LIN {X 0,Y 122.403,Z 271.681,A -85,B 0,C 180,E1 -25569.931,E2 -25569.931} C_VEL
LIN {X 0,Y 122.203,Z 271.74,A -85,B 0,C 180,E1 -25573.312,E2 -25573.312} C_VEL
LIN {X 0,Y 122.006,Z 271.743,A -85,B 0,C 180,E1 -25580.233,E2 -25580.233} C_VEL
LIN {X 0,Y 121.968,Z 271.772,A -85,B 0,C 180,E1 -25583.801,E2 -25583.801} C_VEL
LIN {X 0,Y 121.949,Z 271.761,A -85,B 0,C 180,E1 -25590.17,E2 -25590.17} C_VEL
LIN {X 0,Y 121.983,Z 272.052,A -85,B 0,C 180,E1 -25592.462,E2 -25592.462} C_VEL
LIN {X 0,Y 122.24,Z 273.019,A -85,B 0,C 180,E1 -25593.12,E2 -25593.12} C_VEL
LIN {X 0,Y 123.846,Z 275.828,A -85,B 0,C 180,E1 -25594.219,E2 -25594.219} C_VEL
LIN {X 0,Y 125.183,Z 277.203,A -85,B 0,C 180,E1 -25594.99,E2 -25594.99} C_VEL
LIN {X 0,Y 127.179,Z 280.419,A -85,B 0,C 180,E1 -25596.188,E2 -25596.188} C_VEL
LIN {X 0,Y 128.715,Z 282.669,A -85,B 0,C 180,E1 -25597.05,E2 -25597.05} C_VEL
LIN {X 0,Y 133.456,Z 290.014,A -85,B 0,C 180,E1 -25599.546,E2 -25599.546} C_VEL
LIN {X 0,Y 138.65,Z 299.249,A -85,B 0,C 180,E1 -25602.083,E2 -25602.083} C_VEL
LIN {X 0,Y 142.571,Z 309.17,A -85,B 0,C 180,E1 -25604.02,E2 -25604.02} C_VEL
LIN {X 0,Y 147.025,Z 322.671,A -85,B 0,C 180,E1 -25606.191,E2 -25606.191} C_VEL
LIN {X 0,Y 147.183,Z 326.823,A -85,B 0,C 180,E1 -25606.489,E2 -25606.489} C_VEL
LIN {X 0,Y 144.077,Z 373.493,A -85,B 0,C 180,E1 -25608.588,E2 -25608.588} C_VEL
LIN {X 0,Y 142.334,Z 386.809,A -85,B 0,C 180,E1 -25609.647,E2 -25609.647} C_VEL
LIN {X 0,Y 140.104,Z 399.24,A -85,B 0,C 180,E1 -25611.163,E2 -25611.163} C_VEL
LIN {X 0,Y 137.46,Z 410.573,A -85,B 0,C 180,E1 -25613.071,E2 -25613.071} C_VEL
LIN {X 0,Y 134.929,Z 419.645,A -85,B 0,C 180,E1 -25615.038,E2 -25615.038} C_VEL
LIN {X 0,Y 131.957,Z 429.601,A -85,B 0,C 180,E1 -25617.813,E2 -25617.813} C_VEL
LIN {X 0,Y 128.677,Z 439.018,A -85,B 0,C 180,E1 -25621.144,E2 -25621.144} C_VEL
LIN {X 0,Y 126.257,Z 446.37,A -85,B 0,C 180,E1 -25624.438,E2 -25624.438} C_VEL
LIN {X 0,Y 123.386,Z 454.68,A -85,B 0,C 180,E1 -25629.14,E2 -25629.14} C_VEL
LIN {X 0,Y 121.564,Z 460.326,A -85,B 0,C 180,E1 -25633.193,E2 -25633.193} C_VEL
LIN {X 0,Y 120.15,Z 465.825,A -85,B 0,C 180,E1 -25638.181,E2 -25638.181} C_VEL
LIN {X 0,Y 119.423,Z 470.097,A -85,B 0,C 180,E1 -25643.235,E2 -25643.235} C_VEL
LIN {X 0,Y 119.243,Z 472.346,A -85,B 0,C 180,E1 -25646.616,E2 -25646.616} C_VEL
LIN {X 0,Y 119.301,Z 474.118,A -85,B 0,C 180,E1 -25649.995,E2 -25649.995} C_VEL
LIN {X 0,Y 119.243,Z 475.435,A -85,B 0,C 180,E1 -25653.374,E2 -25653.374} C_VEL
LIN {X 0,Y 119.973,Z 476.91,A -85,B 0,C 180,E1 -25660.116,E2 -25660.116} C_VEL
LIN {X 0,Y 120.788,Z 477.062,A -85,B 0,C 180,E1 -25663.453,E2 -25663.453} C_VEL
LIN {X 0,Y 123.519,Z 476.182,A -85,B 0,C 180,E1 -25669.956,E2 -25669.956} C_VEL
LIN {X 0,Y 127.871,Z 473.795,A -85,B 0,C 180,E1 -25676.079,E2 -25676.079} C_VEL
LIN {X 0,Y 132.095,Z 470.901,A -85,B 0,C 180,E1 -25680.355,E2 -25680.355} C_VEL
LIN {X 0,Y 137.033,Z 466.958,A -85,B 0,C 180,E1 -25684.4,E2 -25684.4} C_VEL
LIN {X 0,Y 142.426,Z 462.037,A -85,B 0,C 180,E1 -25688.078,E2 -25688.078} C_VEL
LIN {X 0,Y 148.475,Z 455.82,A -85,B 0,C 180,E1 -25691.499,E2 -25691.499} C_VEL
LIN {X 0,Y 152.037,Z 451.846,A -85,B 0,C 180,E1 -25693.187,E2 -25693.187} C_VEL
LIN {X 0,Y 153.514,Z 449.546,A -85,B 0,C 180,E1 -25694.277,E2 -25694.277} C_VEL
LIN {X 0,Y 155.933,Z 442.183,A -85,B 0,C 180,E1 -25698.383,E2 -25698.383} C_VEL
LIN {X 0,Y 157.534,Z 439.51,A -85,B 0,C 180,E1 -25699.288,E2 -25699.288} C_VEL
LIN {X 0,Y 163.973,Z 429.783,A -85,B 0,C 180,E1 -25701.456,E2 -25701.456} C_VEL
LIN {X 0,Y 170.017,Z 419.002,A -85,B 0,C 180,E1 -25703.21,E2 -25703.21} C_VEL
LIN {X 0,Y 175.47,Z 406.794,A -85,B 0,C 180,E1 -25704.686,E2 -25704.686} C_VEL
LIN {X 0,Y 179.465,Z 395.485,A -85,B 0,C 180,E1 -25705.679,E2 -25705.679} C_VEL
LIN {X 0,Y 182.83,Z 382.797,A -85,B 0,C 180,E1 -25706.459,E2 -25706.459} C_VEL
LIN {X 0,Y 185.096,Z 369.4,A -85,B 0,C 180,E1 -25706.986,E2 -25706.986} C_VEL
LIN {X 0,Y 186.027,Z 359.421,A -85,B 0,C 180,E1 -25707.359,E2 -25707.359} C_VEL
LIN {X 0,Y 183.427,Z 352.397,A -85,B 0,C 180,E1 -25710.038,E2 -25710.038} C_VEL
LIN {X 0,Y 180.664,Z 345.623,A -85,B 0,C 180,E1 -25713.403,E2 -25713.403} C_VEL
LIN {X 0,Y 178.531,Z 341.006,A -85,B 0,C 180,E1 -25716.548,E2 -25716.548} C_VEL
LIN {X 0,Y 177.003,Z 337.999,A -85,B 0,C 180,E1 -25719.316,E2 -25719.316} C_VEL
LIN {X 0,Y 175.209,Z 334.802,A -85,B 0,C 180,E1 -25724.285,E2 -25724.285} C_VEL
LIN {X 0,Y 174.993,Z 333.83,A -85,B 0,C 180,E1 -25725.558,E2 -25725.558} C_VEL
LIN {X 0,Y 174.576,Z 333.513,A -85,B 0,C 180,E1 -25730.725,E2 -25730.725} C_VEL
LIN {X 0,Y 175.407,Z 334.052,A -85,B 0,C 180,E1 -25735.276,E2 -25735.276} C_VEL
LIN {X 0,Y 176.87,Z 337.493,A -85,B 0,C 180,E1 -25739.595,E2 -25739.595} C_VEL
LIN {X 0,Y 177.65,Z 338.721,A -85,B 0,C 180,E1 -25741.069,E2 -25741.069} C_VEL
LIN {X 0,Y 179.573,Z 342.304,A -85,B 0,C 180,E1 -25744.164,E2 -25744.164} C_VEL
LIN {X 0,Y 182.057,Z 347.068,A -85,B 0,C 180,E1 -25747.381,E2 -25747.381} C_VEL
LIN {X 0,Y 184.322,Z 352.16,A -85,B 0,C 180,E1 -25749.883,E2 -25749.883} C_VEL
LIN {X 0,Y 186.256,Z 356.945,A -85,B 0,C 180,E1 -25751.795,E2 -25751.795} C_VEL
LIN {X 0,Y 184.328,Z 373.568,A -85,B 0,C 180,E1 -25752.362,E2 -25752.362} C_VEL
LIN {X 0,Y 181.73,Z 386.098,A -85,B 0,C 180,E1 -25752.999,E2 -25752.999} C_VEL
LIN {X 0,Y 177.786,Z 399.152,A -85,B 0,C 180,E1 -25753.996,E2 -25753.996} C_VEL
LIN {X 0,Y 173.022,Z 411.143,A -85,B 0,C 180,E1 -25755.284,E2 -25755.284} C_VEL
LIN {X 0,Y 167.29,Z 422.614,A -85,B 0,C 180,E1 -25756.966,E2 -25756.966} C_VEL
LIN {X 0,Y 160.799,Z 433.232,A -85,B 0,C 180,E1 -25759.076,E2 -25759.076} C_VEL
LIN {X 0,Y 154.773,Z 441.601,A -85,B 0,C 180,E1 -25761.289,E2 -25761.289} C_VEL
LIN {X 0,Y 148.126,Z 449.538,A -85,B 0,C 180,E1 -25764.041,E2 -25764.041} C_VEL
LIN {X 0,Y 140.778,Z 457.024,A -85,B 0,C 180,E1 -25767.62,E2 -25767.62} C_VEL
LIN {X 0,Y 134.12,Z 462.882,A -85,B 0,C 180,E1 -25771.587,E2 -25771.587} C_VEL
LIN {X 0,Y 127.366,Z 467.973,A -85,B 0,C 180,E1 -25776.642,E2 -25776.642} C_VEL
LIN {X 0,Y 122.243,Z 471.149,A -85,B 0,C 180,E1 -25781.643,E2 -25781.643} C_VEL
LIN {X 0,Y 119.474,Z 472.56,A -85,B 0,C 180,E1 -25785.106,E2 -25785.106} C_VEL
LIN {X 0,Y 117.087,Z 473.521,A -85,B 0,C 180,E1 -25788.688,E2 -25788.688} C_VEL
LIN {X 0,Y 115.063,Z 473.981,A -85,B 0,C 180,E1 -25792.539,E2 -25792.539} C_VEL
LIN {X 0,Y 113.602,Z 473.972,A -85,B 0,C 180,E1 -25796.173,E2 -25796.173} C_VEL
LIN {X 0,Y 112.308,Z 473.302,A -85,B 0,C 180,E1 -25801.141,E2 -25801.141} C_VEL
LIN {X 0,Y 111.542,Z 471.221,A -85,B 0,C 180,E1 -25807.794,E2 -25807.794} C_VEL
LIN {X 0,Y 111.803,Z 468.27,A -85,B 0,C 180,E1 -25813.574,E2 -25813.574} C_VEL
LIN {X 0,Y 112.709,Z 464.215,A -85,B 0,C 180,E1 -25819.224,E2 -25819.224} C_VEL
LIN {X 0,Y 114.241,Z 458.968,A -85,B 0,C 180,E1 -25824.711,E2 -25824.711} C_VEL
LIN {X 0,Y 116.441,Z 452.342,A -85,B 0,C 180,E1 -25830.005,E2 -25830.005} C_VEL
LIN {X 0,Y 119.479,Z 444.069,A -85,B 0,C 180,E1 -25835.045,E2 -25835.045} C_VEL
LIN {X 0,Y 122.529,Z 435.547,A -85,B 0,C 180,E1 -25839.081,E2 -25839.081} C_VEL
LIN {X 0,Y 125.838,Z 426.24,A -85,B 0,C 180,E1 -25842.504,E2 -25842.504} C_VEL
LIN {X 0,Y 129.091,Z 416.094,A -85,B 0,C 180,E1 -25845.396,E2 -25845.396} C_VEL
LIN {X 0,Y 132.092,Z 405.057,A -85,B 0,C 180,E1 -25847.819,E2 -25847.819} C_VEL
LIN {X 0,Y 134.949,Z 392.373,A -85,B 0,C 180,E1 -25849.878,E2 -25849.878} C_VEL
LIN {X 0,Y 137.118,Z 379.343,A -85,B 0,C 180,E1 -25851.348,E2 -25851.348} C_VEL
LIN {X 0,Y 138.593,Z 365.838,A -85,B 0,C 180,E1 -25852.288,E2 -25852.288} C_VEL
LIN {X 0,Y 141.572,Z 321.306,A -85,B 0,C 180,E1 -25854.321,E2 -25854.321} C_VEL
LIN {X 0,Y 138.053,Z 311.535,A -85,B 0,C 180,E1 -25856.101,E2 -25856.101} C_VEL
LIN {X 0,Y 133.083,Z 301.541,A -85,B 0,C 180,E1 -25858.579,E2 -25858.579} C_VEL
LIN {X 0,Y 126.471,Z 290.227,A -85,B 0,C 180,E1 -25862.157,E2 -25862.157} C_VEL
LIN {X 0,Y 120.762,Z 281.835,A -85,B 0,C 180,E1 -25865.641,E2 -25865.641} C_VEL
LIN {X 0,Y 118.642,Z 278.829,A -85,B 0,C 180,E1 -25867.062,E2 -25867.062} C_VEL
LIN {X 0,Y 117.859,Z 277.647,A -85,B 0,C 180,E1 -25867.618,E2 -25867.618} C_VEL
LIN {X 0,Y 115.795,Z 275.519,A -85,B 0,C 180,E1 -25869.05,E2 -25869.05} C_VEL
LIN {X 0,Y 114.906,Z 273.28,A -85,B 0,C 180,E1 -25870.113,E2 -25870.113} C_VEL
LIN {X 0,Y 114.82,Z 272.739,A -85,B 0,C 180,E1 -25871.018,E2 -25871.018} C_VEL
LIN {X 0,Y 114.755,Z 272.648,A -85,B 0,C 180,E1 -25877.669,E2 -25877.669} C_VEL
LIN {X 0,Y 114.771,Z 272.671,A -85,B 0,C 180,E1 -25882.763,E2 -25882.763} C_VEL
LIN {X 0,Y 114.83,Z 272.625,A -85,B 0,C 180,E1 -25888.975,E2 -25888.975} C_VEL
LIN {X 0,Y 114.896,Z 272.673,A -85,B 0,C 180,E1 -25896.58,E2 -25896.58} C_VEL
LIN {X 0,Y 114.965,Z 272.598,A -85,B 0,C 180,E1 -25902.217,E2 -25902.217} C_VEL
LIN {X 0,Y 115.31,Z 272.62,A -85,B 0,C 180,E1 -25909.479,E2 -25909.479} C_VEL
LIN {X 0,Y 115.487,Z 272.532,A -85,B 0,C 180,E1 -25916.525,E2 -25916.525} C_VEL
LIN {X 0,Y 115.956,Z 272.498,A -85,B 0,C 180,E1 -25920.013,E2 -25920.013} C_VEL
LIN {X 0,Y 115.356,Z 272.57,A -85,B 0,C 180,E1 -25927.012,E2 -25927.012} C_VEL
LIN {X 0,Y 115.219,Z 272.595,A -85,B 0,C 180,E1 -25932.568,E2 -25932.568} C_VEL
LIN {X 0,Y 114.983,Z 272.632,A -85,B 0,C 180,E1 -25937.808,E2 -25937.808} C_VEL
LIN {X 0,Y 114.931,Z 272.641,A -85,B 0,C 180,E1 -25943.461,E2 -25943.461} C_VEL
LIN {X 0,Y 114.904,Z 272.908,A -85,B 0,C 180,E1 -25948.372,E2 -25948.372} C_VEL
LIN {X 0,Y 115.209,Z 274.1,A -85,B 0,C 180,E1 -25949.225,E2 -25949.225} C_VEL
LIN {X 0,Y 116.985,Z 276.842,A -85,B 0,C 180,E1 -25950.626,E2 -25950.626} C_VEL
LIN {X 0,Y 118.483,Z 278.361,A -85,B 0,C 180,E1 -25951.635,E2 -25951.635} C_VEL
LIN {X 0,Y 120.642,Z 281.71,A -85,B 0,C 180,E1 -25953.117,E2 -25953.117} C_VEL
LIN {X 0,Y 121.817,Z 283.352,A -85,B 0,C 180,E1 -25953.869,E2 -25953.869} C_VEL
LIN {X 0,Y 126.872,Z 290.91,A -85,B 0,C 180,E1 -25956.905,E2 -25956.905} C_VEL
LIN {X 0,Y 133.463,Z 302.405,A -85,B 0,C 180,E1 -25960.457,E2 -25960.457} C_VEL
LIN {X 0,Y 137.115,Z 311.613,A -85,B 0,C 180,E1 -25962.416,E2 -25962.416} C_VEL
LIN {X 0,Y 141.44,Z 325.033,A -85,B 0,C 180,E1 -25964.709,E2 -25964.709} C_VEL
LIN {X 0,Y 138.165,Z 373.629,A -85,B 0,C 180,E1 -25966.999,E2 -25966.999} C_VEL
LIN {X 0,Y 136.379,Z 386.631,A -85,B 0,C 180,E1 -25968.057,E2 -25968.057} C_VEL
LIN {X 0,Y 134.123,Z 398.758,A -85,B 0,C 180,E1 -25969.57,E2 -25969.57} C_VEL
LIN {X 0,Y 131.352,Z 410.199,A -85,B 0,C 180,E1 -25971.532,E2 -25971.532} C_VEL
LIN {X 0,Y 128.697,Z 419.304,A -85,B 0,C 180,E1 -25973.562,E2 -25973.562} C_VEL
LIN {X 0,Y 125.567,Z 429.32,A -85,B 0,C 180,E1 -25976.442,E2 -25976.442} C_VEL
LIN {X 0,Y 122.067,Z 438.887,A -85,B 0,C 180,E1 -25979.962,E2 -25979.962} C_VEL
LIN {X 0,Y 119.873,Z 445.38,A -85,B 0,C 180,E1 -25982.97,E2 -25982.97} C_VEL
LIN {X 0,Y 116.755,Z 453.855,A -85,B 0,C 180,E1 -25987.895,E2 -25987.895} C_VEL
LIN {X 0,Y 114.441,Z 460.654,A -85,B 0,C 180,E1 -25993.034,E2 -25993.034} C_VEL
LIN {X 0,Y 112.818,Z 466.865,A -85,B 0,C 180,E1 -25999.223,E2 -25999.223} C_VEL
LIN {X 0,Y 112.212,Z 470.866,A -85,B 0,C 180,E1 -26004.604,E2 -26004.604} C_VEL
LIN {X 0,Y 112.22,Z 473.796,A -85,B 0,C 180,E1 -26009.994,E2 -26009.994} C_VEL
LIN {X 0,Y 112.154,Z 475.171,A -85,B 0,C 180,E1 -26013.587,E2 -26013.587} C_VEL
LIN {X 0,Y 112.972,Z 476.74,A -85,B 0,C 180,E1 -26020.75,E2 -26020.75} C_VEL
LIN {X 0,Y 115.178,Z 476.779,A -85,B 0,C 180,E1 -26027.758,E2 -26027.758} C_VEL
LIN {X 0,Y 118.965,Z 475.247,A -85,B 0,C 180,E1 -26034.421,E2 -26034.421} C_VEL
LIN {X 0,Y 124.442,Z 472.172,A -85,B 0,C 180,E1 -26040.543,E2 -26040.543} C_VEL
LIN {X 0,Y 129.381,Z 468.73,A -85,B 0,C 180,E1 -26044.769,E2 -26044.769} C_VEL
LIN {X 0,Y 134.895,Z 464.25,A -85,B 0,C 180,E1 -26048.69,E2 -26048.69} C_VEL
LIN {X 0,Y 142.17,Z 457.507,A -85,B 0,C 180,E1 -26052.815,E2 -26052.815} C_VEL
LIN {X 0,Y 149.058,Z 450.213,A -85,B 0,C 180,E1 -26055.968,E2 -26055.968} C_VEL
LIN {X 0,Y 156.292,Z 441.211,A -85,B 0,C 180,E1 -26058.862,E2 -26058.862} C_VEL
LIN {X 0,Y 157.534,Z 439.51,A -85,B 0,C 180,E1 -26059.288,E2 -26059.288} C_VEL
LIN {X 0,Y 160.137,Z 435.355,A -85,B 0,C 180,E1 -26060.469,E2 -26060.469} C_VEL
LIN {X 0,Y 163.166,Z 428.411,A -85,B 0,C 180,E1 -26062.738,E2 -26062.738} C_VEL
LIN {X 0,Y 165.973,Z 421.086,A -85,B 0,C 180,E1 -26064.83,E2 -26064.83} C_VEL
LIN {X 0,Y 168.136,Z 416.223,A -85,B 0,C 180,E1 -26065.725,E2 -26065.725} C_VEL
LIN {X 0,Y 172.963,Z 405.394,A -85,B 0,C 180,E1 -26066.928,E2 -26066.928} C_VEL
LIN {X 0,Y 177.071,Z 393.675,A -85,B 0,C 180,E1 -26067.893,E2 -26067.893} C_VEL
LIN {X 0,Y 180.496,Z 380.166,A -85,B 0,C 180,E1 -26068.636,E2 -26068.636} C_VEL
LIN {X 0,Y 182.557,Z 367.334,A -85,B 0,C 180,E1 -26069.081,E2 -26069.081} C_VEL
LIN {X 0,Y 182.952,Z 362.799,A -85,B 0,C 180,E1 -26069.275,E2 -26069.275} C_VEL
LIN {X 0,Y 180.739,Z 356.713,A -85,B 0,C 180,E1 -26071.861,E2 -26071.861} C_VEL
LIN {X 0,Y 178.612,Z 351.184,A -85,B 0,C 180,E1 -26074.814,E2 -26074.814} C_VEL
LIN {X 0,Y 176.995,Z 347.376,A -85,B 0,C 180,E1 -26077.474,E2 -26077.474} C_VEL
LIN {X 0,Y 175.737,Z 344.777,A -85,B 0,C 180,E1 -26079.952,E2 -26079.952} C_VEL
LIN {X 0,Y 174.126,Z 341.381,A -85,B 0,C 180,E1 -26085.119,E2 -26085.119} C_VEL
LIN {X 0,Y 174.003,Z 340.799,A -85,B 0,C 180,E1 -26085.967,E2 -26085.967} C_VEL
LIN {X 0,Y 173.971,Z 340.663,A -85,B 0,C 180,E1 -26093.03,E2 -26093.03} C_VEL
LIN {X 0,Y 174.388,Z 341.072,A -85,B 0,C 180,E1 -26094.918,E2 -26094.918} C_VEL
LIN {X 0,Y 175.915,Z 344.609,A -85,B 0,C 180,E1 -26099.558,E2 -26099.558} C_VEL
LIN {X 0,Y 177.962,Z 348.626,A -85,B 0,C 180,E1 -26103.247,E2 -26103.247} C_VEL
LIN {X 0,Y 180.32,Z 353.423,A -85,B 0,C 180,E1 -26106.543,E2 -26106.543} C_VEL
LIN {X 0,Y 182.873,Z 359.659,A -85,B 0,C 180,E1 -26109.56,E2 -26109.56} C_VEL
LIN {X 0,Y 183.179,Z 360.526,A -85,B 0,C 180,E1 -26109.895,E2 -26109.895} C_VEL
LIN {X 0,Y 181.29,Z 375.016,A -85,B 0,C 180,E1 -26110.377,E2 -26110.377} C_VEL
LIN {X 0,Y 178.531,Z 387.326,A -85,B 0,C 180,E1 -26111.007,E2 -26111.007} C_VEL
LIN {X 0,Y 174.297,Z 400.567,A -85,B 0,C 180,E1 -26112.018,E2 -26112.018} C_VEL
LIN {X 0,Y 169.637,Z 411.763,A -85,B 0,C 180,E1 -26113.214,E2 -26113.214} C_VEL
LIN {X 0,Y 163.996,Z 422.64,A -85,B 0,C 180,E1 -26114.776,E2 -26114.776} C_VEL
LIN {X 0,Y 157.001,Z 433.645,A -85,B 0,C 180,E1 -26116.912,E2 -26116.912} C_VEL
LIN {X 0,Y 150.367,Z 442.437,A -85,B 0,C 180,E1 -26119.231,E2 -26119.231} C_VEL
LIN {X 0,Y 143.809,Z 449.846,A -85,B 0,C 180,E1 -26121.806,E2 -26121.806} C_VEL
LIN {X 0,Y 136.11,Z 457.281,A -85,B 0,C 180,E1 -26125.375,E2 -26125.375} C_VEL
LIN {X 0,Y 129.035,Z 463.133,A -85,B 0,C 180,E1 -26129.383,E2 -26129.383} C_VEL
LIN {X 0,Y 122.695,Z 467.622,A -85,B 0,C 180,E1 -26133.853,E2 -26133.853} C_VEL
LIN {X 0,Y 117.172,Z 470.875,A -85,B 0,C 180,E1 -26138.772,E2 -26138.772} C_VEL
LIN {X 0,Y 113.581,Z 472.578,A -85,B 0,C 180,E1 -26142.873,E2 -26142.873} C_VEL
LIN {X 0,Y 109.052,Z 474.029,A -85,B 0,C 180,E1 -26149.883,E2 -26149.883} C_VEL
LIN {X 0,Y 107.247,Z 474.118,A -85,B 0,C 180,E1 -26153.866,E2 -26153.866} C_VEL
LIN {X 0,Y 105.372,Z 473.395,A -85,B 0,C 180,E1 -26160.086,E2 -26160.086} C_VEL
LIN {X 0,Y 104.506,Z 471.675,A -85,B 0,C 180,E1 -26166.21,E2 -26166.21} C_VEL
LIN {X 0,Y 104.569,Z 468.88,A -85,B 0,C 180,E1 -26172.402,E2 -26172.402} C_VEL
LIN {X 0,Y 105.427,Z 464.981,A -85,B 0,C 180,E1 -26178.47,E2 -26178.47} C_VEL
LIN {X 0,Y 106.943,Z 459.901,A -85,B 0,C 180,E1 -26184.349,E2 -26184.349} C_VEL
LIN {X 0,Y 109.072,Z 453.516,A -85,B 0,C 180,E1 -26190.006,E2 -26190.006} C_VEL
LIN {X 0,Y 112.176,Z 445.493,A -85,B 0,C 180,E1 -26195.4,E2 -26195.4} C_VEL
LIN {X 0,Y 115.39,Z 437.259,A -85,B 0,C 180,E1 -26199.647,E2 -26199.647} C_VEL
LIN {X 0,Y 119.136,Z 427.186,A -85,B 0,C 180,E1 -26203.654,E2 -26203.654} C_VEL
LIN {X 0,Y 122.515,Z 417.27,A -85,B 0,C 180,E1 -26206.673,E2 -26206.673} C_VEL
LIN {X 0,Y 125.684,Z 406.532,A -85,B 0,C 180,E1 -26209.184,E2 -26209.184} C_VEL
LIN {X 0,Y 128.518,Z 394.802,A -85,B 0,C 180,E1 -26211.235,E2 -26211.235} C_VEL
LIN {X 0,Y 131.06,Z 381.118,A -85,B 0,C 180,E1 -26212.921,E2 -26212.921} C_VEL
LIN {X 0,Y 132.678,Z 367.926,A -85,B 0,C 180,E1 -26213.93,E2 -26213.93} C_VEL
LIN {X 0,Y 135.961,Z 323.313,A -85,B 0,C 180,E1 -26215.99,E2 -26215.99} C_VEL
LIN {X 0,Y 132.938,Z 314.805,A -85,B 0,C 180,E1 -26217.661,E2 -26217.661} C_VEL
LIN {X 0,Y 128.25,Z 305.355,A -85,B 0,C 180,E1 -26220.189,E2 -26220.189} C_VEL
LIN {X 0,Y 122.378,Z 295.105,A -85,B 0,C 180,E1 -26223.653,E2 -26223.653} C_VEL
LIN {X 0,Y 117.429,Z 287.522,A -85,B 0,C 180,E1 -26226.913,E2 -26226.913} C_VEL
LIN {X 0,Y 114.355,Z 283.287,A -85,B 0,C 180,E1 -26229.148,E2 -26229.148} C_VEL
LIN {X 0,Y 112.028,Z 280.176,A -85,B 0,C 180,E1 -26230.99,E2 -26230.99} C_VEL
LIN {X 0,Y 111.299,Z 278.889,A -85,B 0,C 180,E1 -26231.635,E2 -26231.635} C_VEL
LIN {X 0,Y 108.763,Z 276.543,A -85,B 0,C 180,E1 -26233.771,E2 -26233.771} C_VEL
LIN {X 0,Y 107.719,Z 274.073,A -85,B 0,C 180,E1 -26235.222,E2 -26235.222} C_VEL
LIN {X 0,Y 107.688,Z 273.578,A -85,B 0,C 180,E1 -26236.77,E2 -26236.77} C_VEL
LIN {X 0,Y 107.699,Z 273.569,A -85,B 0,C 180,E1 -26244.053,E2 -26244.053} C_VEL
LIN {X 0,Y 107.768,Z 273.505,A -85,B 0,C 180,E1 -26248.571,E2 -26248.571} C_VEL
LIN {X 0,Y 107.863,Z 273.548,A -85,B 0,C 180,E1 -26257.004,E2 -26257.004} C_VEL
LIN {X 0,Y 107.86,Z 273.489,A -85,B 0,C 180,E1 -26261.003,E2 -26261.003} C_VEL
LIN {X 0,Y 108.228,Z 273.495,A -85,B 0,C 180,E1 -26268.781,E2 -26268.781} C_VEL
LIN {X 0,Y 108.291,Z 273.46,A -85,B 0,C 180,E1 -26272.557,E2 -26272.557} C_VEL
LIN {X 0,Y 108.886,Z 273.375,A -85,B 0,C 180,E1 -26280.014,E2 -26280.014} C_VEL
LIN {X 0,Y 108.297,Z 273.443,A -85,B 0,C 180,E1 -26287.472,E2 -26287.472} C_VEL
LIN {X 0,Y 108.153,Z 273.477,A -85,B 0,C 180,E1 -26292.884,E2 -26292.884} C_VEL
LIN {X 0,Y 107.897,Z 273.498,A -85,B 0,C 180,E1 -26301.007,E2 -26301.007} C_VEL
LIN {X 0,Y 107.937,Z 273.848,A -85,B 0,C 180,E1 -26303.567,E2 -26303.567} C_VEL
LIN {X 0,Y 108.215,Z 275.116,A -85,B 0,C 180,E1 -26304.432,E2 -26304.432} C_VEL
LIN {X 0,Y 109.831,Z 277.695,A -85,B 0,C 180,E1 -26305.995,E2 -26305.995} C_VEL
LIN {X 0,Y 111.72,Z 279.308,A -85,B 0,C 180,E1 -26307.529,E2 -26307.529} C_VEL
LIN {X 0,Y 113.783,Z 282.572,A -85,B 0,C 180,E1 -26309.246,E2 -26309.246} C_VEL
LIN {X 0,Y 115.207,Z 284.265,A -85,B 0,C 180,E1 -26310.304,E2 -26310.304} C_VEL
LIN {X 0,Y 120.719,Z 292.539,A -85,B 0,C 180,E1 -26314.133,E2 -26314.133} C_VEL
LIN {X 0,Y 125.969,Z 301.247,A -85,B 0,C 180,E1 -26317.345,E2 -26317.345} C_VEL
LIN {X 0,Y 129.654,Z 308.507,A -85,B 0,C 180,E1 -26319.45,E2 -26319.45} C_VEL
LIN {X 0,Y 133.071,Z 318.038,A -85,B 0,C 180,E1 -26321.451,E2 -26321.451} C_VEL
LIN {X 0,Y 135.778,Z 326.645,A -85,B 0,C 180,E1 -26323.008,E2 -26323.008} C_VEL
LIN {X 0,Y 132.451,Z 373.031,A -85,B 0,C 180,E1 -26325.218,E2 -26325.218} C_VEL
LIN {X 0,Y 130.604,Z 386.006,A -85,B 0,C 180,E1 -26326.273,E2 -26326.273} C_VEL
LIN {X 0,Y 128.036,Z 399.42,A -85,B 0,C 180,E1 -26328.005,E2 -26328.005} C_VEL
LIN {X 0,Y 124.845,Z 411.421,A -85,B 0,C 180,E1 -26330.177,E2 -26330.177} C_VEL
LIN {X 0,Y 122.153,Z 420.348,A -85,B 0,C 180,E1 -26332.31,E2 -26332.31} C_VEL
LIN {X 0,Y 118.889,Z 430.129,A -85,B 0,C 180,E1 -26335.315,E2 -26335.315} C_VEL
LIN {X 0,Y 115.016,Z 440.25,A -85,B 0,C 180,E1 -26339.33,E2 -26339.33} C_VEL
LIN {X 0,Y 112.267,Z 447.423,A -85,B 0,C 180,E1 -26343.003,E2 -26343.003} C_VEL
LIN {X 0,Y 109.178,Z 455.518,A -85,B 0,C 180,E1 -26348.27,E2 -26348.27} C_VEL
LIN {X 0,Y 107.303,Z 460.981,A -85,B 0,C 180,E1 -26352.852,E2 -26352.852} C_VEL
LIN {X 0,Y 105.838,Z 466.306,A -85,B 0,C 180,E1 -26358.503,E2 -26358.503} C_VEL
LIN {X 0,Y 105.134,Z 470.415,A -85,B 0,C 180,E1 -26364.239,E2 -26364.239} C_VEL
LIN {X 0,Y 105.128,Z 473.439,A -85,B 0,C 180,E1 -26369.994,E2 -26369.994} C_VEL
LIN {X 0,Y 105.089,Z 474.905,A -85,B 0,C 180,E1 -26373.829,E2 -26373.829} C_VEL
LIN {X 0,Y 105.998,Z 476.57,A -85,B 0,C 180,E1 -26381.467,E2 -26381.467} C_VEL
LIN {X 0,Y 108.428,Z 476.73,A -85,B 0,C 180,E1 -26388.904,E2 -26388.904} C_VEL
LIN {X 0,Y 110.223,Z 476.219,A -85,B 0,C 180,E1 -26392.487,E2 -26392.487} C_VEL
LIN {X 0,Y 115.286,Z 474.03,A -85,B 0,C 180,E1 -26399.183,E2 -26399.183} C_VEL
LIN {X 0,Y 120.028,Z 471.342,A -85,B 0,C 180,E1 -26403.79,E2 -26403.79} C_VEL
LIN {X 0,Y 126.973,Z 466.639,A -85,B 0,C 180,E1 -26408.983,E2 -26408.983} C_VEL
LIN {X 0,Y 133.696,Z 461.136,A -85,B 0,C 180,E1 -26413.101,E2 -26413.101} C_VEL
LIN {X 0,Y 140.591,Z 454.726,A -85,B 0,C 180,E1 -26416.449,E2 -26416.449} C_VEL
LIN {X 0,Y 147.978,Z 446.776,A -85,B 0,C 180,E1 -26419.448,E2 -26419.448} C_VEL
LIN {X 0,Y 154.41,Z 438.703,A -85,B 0,C 180,E1 -26421.726,E2 -26421.726} C_VEL
LIN {X 0,Y 160.385,Z 429.953,A -85,B 0,C 180,E1 -26423.621,E2 -26423.621} C_VEL
LIN {X 0,Y 166.618,Z 419.248,A -85,B 0,C 180,E1 -26425.33,E2 -26425.33} C_VEL
LIN {X 0,Y 168.136,Z 416.223,A -85,B 0,C 180,E1 -26425.725,E2 -26425.725} C_VEL
LIN {X 0,Y 170.201,Z 411.242,A -85,B 0,C 180,E1 -26426.557,E2 -26426.557} C_VEL
LIN {X 0,Y 172.468,Z 403.032,A -85,B 0,C 180,E1 -26428.27,E2 -26428.27} C_VEL
LIN {X 0,Y 174.356,Z 394.49,A -85,B 0,C 180,E1 -26429.785,E2 -26429.785} C_VEL
LIN {X 0,Y 175.74,Z 389.002,A -85,B 0,C 180,E1 -26430.31,E2 -26430.31} C_VEL
LIN {X 0,Y 178.689,Z 376.276,A -85,B 0,C 180,E1 -26430.885,E2 -26430.885} C_VEL
LIN {X 0,Y 180.094,Z 366.402,A -85,B 0,C 180,E1 -26431.24,E2 -26431.24} C_VEL
LIN {X 0,Y 177.797,Z 359.666,A -85,B 0,C 180,E1 -26434.454,E2 -26434.454} C_VEL
LIN {X 0,Y 175.986,Z 354.801,A -85,B 0,C 180,E1 -26437.514,E2 -26437.514} C_VEL
LIN {X 0,Y 174.551,Z 351.613,A -85,B 0,C 180,E1 -26440.507,E2 -26440.507} C_VEL
LIN {X 0,Y 173.085,Z 348.039,A -85,B 0,C 180,E1 -26445.891,E2 -26445.891} C_VEL
LIN {X 0,Y 172.783,Z 347.621,A -85,B 0,C 180,E1 -26448.257,E2 -26448.257} C_VEL
LIN {X 0,Y 173.294,Z 347.843,A -85,B 0,C 180,E1 -26454.131,E2 -26454.131} C_VEL
LIN {X 0,Y 175.111,Z 352.223,A -85,B 0,C 180,E1 -26459.882,E2 -26459.882} C_VEL
LIN {X 0,Y 176.701,Z 355.665,A -85,B 0,C 180,E1 -26462.837,E2 -26462.837} C_VEL
LIN {X 0,Y 178.814,Z 360.162,A -85,B 0,C 180,E1 -26465.943,E2 -26465.943} C_VEL
LIN {X 0,Y 180.259,Z 364.22,A -85,B 0,C 180,E1 -26467.874,E2 -26467.874} C_VEL
LIN {X 0,Y 178.452,Z 376.563,A -85,B 0,C 180,E1 -26468.337,E2 -26468.337} C_VEL
LIN {X 0,Y 175.037,Z 390.351,A -85,B 0,C 180,E1 -26469.069,E2 -26469.069} C_VEL
LIN {X 0,Y 170.819,Z 402.508,A -85,B 0,C 180,E1 -26470.008,E2 -26470.008} C_VEL
LIN {X 0,Y 165.691,Z 413.914,A -85,B 0,C 180,E1 -26471.245,E2 -26471.245} C_VEL
LIN {X 0,Y 159.642,Z 424.797,A -85,B 0,C 180,E1 -26472.847,E2 -26472.847} C_VEL
LIN {X 0,Y 152.692,Z 435.097,A -85,B 0,C 180,E1 -26474.875,E2 -26474.875} C_VEL
LIN {X 0,Y 145.379,Z 444.109,A -85,B 0,C 180,E1 -26477.315,E2 -26477.315} C_VEL
LIN {X 0,Y 136.98,Z 452.806,A -85,B 0,C 180,E1 -26480.568,E2 -26480.568} C_VEL
LIN {X 0,Y 129.089,Z 459.65,A -85,B 0,C 180,E1 -26484.241,E2 -26484.241} C_VEL
LIN {X 0,Y 122.56,Z 464.524,A -85,B 0,C 180,E1 -26488,E2 -26488} C_VEL
LIN {X 0,Y 115.143,Z 469.132,A -85,B 0,C 180,E1 -26493.304,E2 -26493.304} C_VEL
LIN {X 0,Y 108.912,Z 472.224,A -85,B 0,C 180,E1 -26499.264,E2 -26499.264} C_VEL
LIN {X 0,Y 105.811,Z 473.351,A -85,B 0,C 180,E1 -26503.07,E2 -26503.07} C_VEL
LIN {X 0,Y 102.012,Z 474.191,A -85,B 0,C 180,E1 -26509.247,E2 -26509.247} C_VEL
LIN {X 0,Y 99.389,Z 473.983,A -85,B 0,C 180,E1 -26515.557,E2 -26515.557} C_VEL
LIN {X 0,Y 98.265,Z 473.27,A -85,B 0,C 180,E1 -26519.965,E2 -26519.965} C_VEL
LIN {X 0,Y 97.543,Z 472.124,A -85,B 0,C 180,E1 -26524.394,E2 -26524.394} C_VEL
LIN {X 0,Y 97.364,Z 470.078,A -85,B 0,C 180,E1 -26529.728,E2 -26529.728} C_VEL
LIN {X 0,Y 97.812,Z 467.098,A -85,B 0,C 180,E1 -26535.442,E2 -26535.442} C_VEL
LIN {X 0,Y 99.224,Z 462.119,A -85,B 0,C 180,E1 -26542.437,E2 -26542.437} C_VEL
LIN {X 0,Y 101.343,Z 455.796,A -85,B 0,C 180,E1 -26549.013,E2 -26549.013} C_VEL
LIN {X 0,Y 104.289,Z 448.301,A -85,B 0,C 180,E1 -26554.838,E2 -26554.838} C_VEL
LIN {X 0,Y 107.623,Z 440.471,A -85,B 0,C 180,E1 -26559.491,E2 -26559.491} C_VEL
LIN {X 0,Y 111.267,Z 431.346,A -85,B 0,C 180,E1 -26563.707,E2 -26563.707} C_VEL
LIN {X 0,Y 115.153,Z 421.026,A -85,B 0,C 180,E1 -26567.315,E2 -26567.315} C_VEL
LIN {X 0,Y 118.842,Z 409.54,A -85,B 0,C 180,E1 -26570.336,E2 -26570.336} C_VEL
LIN {X 0,Y 122.083,Z 397.55,A -85,B 0,C 180,E1 -26572.667,E2 -26572.667} C_VEL
LIN {X 0,Y 124.801,Z 384.618,A -85,B 0,C 180,E1 -26574.431,E2 -26574.431} C_VEL
LIN {X 0,Y 126.784,Z 370.797,A -85,B 0,C 180,E1 -26575.662,E2 -26575.662} C_VEL
LIN {X 0,Y 130.338,Z 324.861,A -85,B 0,C 180,E1 -26577.888,E2 -26577.888} C_VEL
LIN {X 0,Y 127.752,Z 317.8,A -85,B 0,C 180,E1 -26579.426,E2 -26579.426} C_VEL
LIN {X 0,Y 122.98,Z 308.092,A -85,B 0,C 180,E1 -26582.262,E2 -26582.262} C_VEL
LIN {X 0,Y 118.236,Z 299.765,A -85,B 0,C 180,E1 -26585.324,E2 -26585.324} C_VEL
LIN {X 0,Y 113.614,Z 292.543,A -85,B 0,C 180,E1 -26588.658,E2 -26588.658} C_VEL
LIN {X 0,Y 110.804,Z 288.558,A -85,B 0,C 180,E1 -26590.905,E2 -26590.905} C_VEL
LIN {X 0,Y 108.167,Z 284.768,A -85,B 0,C 180,E1 -26593.246,E2 -26593.246} C_VEL
LIN {X 0,Y 105.657,Z 281.989,A -85,B 0,C 180,E1 -26595.585,E2 -26595.585} C_VEL
LIN {X 0,Y 104.713,Z 280.046,A -85,B 0,C 180,E1 -26596.654,E2 -26596.654} C_VEL
LIN {X 0,Y 101.89,Z 277.693,A -85,B 0,C 180,E1 -26599.675,E2 -26599.675} C_VEL
LIN {X 0,Y 100.731,Z 275.009,A -85,B 0,C 180,E1 -26601.763,E2 -26601.763} C_VEL
LIN {X 0,Y 100.653,Z 274.475,A -85,B 0,C 180,E1 -26603.615,E2 -26603.615} C_VEL
LIN {X 0,Y 100.672,Z 274.403,A -85,B 0,C 180,E1 -26606.912,E2 -26606.912} C_VEL
LIN {X 0,Y 100.721,Z 274.422,A -85,B 0,C 180,E1 -26615.268,E2 -26615.268} C_VEL
LIN {X 0,Y 100.774,Z 274.384,A -85,B 0,C 180,E1 -26619.609,E2 -26619.609} C_VEL
LIN {X 0,Y 101.127,Z 274.36,A -85,B 0,C 180,E1 -26627.982,E2 -26627.982} C_VEL
LIN {X 0,Y 101.228,Z 274.344,A -85,B 0,C 180,E1 -26632.034,E2 -26632.034} C_VEL
LIN {X 0,Y 101.817,Z 274.252,A -85,B 0,C 180,E1 -26640.015,E2 -26640.015} C_VEL
LIN {X 0,Y 101.232,Z 274.317,A -85,B 0,C 180,E1 -26647.997,E2 -26647.997} C_VEL
LIN {X 0,Y 101.024,Z 274.382,A -85,B 0,C 180,E1 -26654.19,E2 -26654.19} C_VEL
LIN {X 0,Y 100.916,Z 274.723,A -85,B 0,C 180,E1 -26656.971,E2 -26656.971} C_VEL
LIN {X 0,Y 101.205,Z 275.903,A -85,B 0,C 180,E1 -26658.094,E2 -26658.094} C_VEL
LIN {X 0,Y 102.866,Z 278.531,A -85,B 0,C 180,E1 -26660.251,E2 -26660.251} C_VEL
LIN {X 0,Y 104.953,Z 280.162,A -85,B 0,C 180,E1 -26662.402,E2 -26662.402} C_VEL
LIN {X 0,Y 106.713,Z 283.28,A -85,B 0,C 180,E1 -26664.277,E2 -26664.277} C_VEL
LIN {X 0,Y 108.88,Z 285.571,A -85,B 0,C 180,E1 -26666.21,E2 -26666.21} C_VEL
LIN {X 0,Y 112.39,Z 290.724,A -85,B 0,C 180,E1 -26669.211,E2 -26669.211} C_VEL
LIN {X 0,Y 116.926,Z 297.608,A -85,B 0,C 180,E1 -26672.598,E2 -26672.598} C_VEL
LIN {X 0,Y 122.07,Z 306.53,A -85,B 0,C 180,E1 -26676.013,E2 -26676.013} C_VEL
LIN {X 0,Y 125.122,Z 312.759,A -85,B 0,C 180,E1 -26677.907,E2 -26677.907} C_VEL
LIN {X 0,Y 128.173,Z 321.75,A -85,B 0,C 180,E1 -26679.875,E2 -26679.875} C_VEL
LIN {X 0,Y 130.173,Z 328.184,A -85,B 0,C 180,E1 -26681.128,E2 -26681.128} C_VEL
LIN {X 0,Y 126.756,Z 373.362,A -85,B 0,C 180,E1 -26683.341,E2 -26683.341} C_VEL
LIN {X 0,Y 124.734,Z 386.929,A -85,B 0,C 180,E1 -26684.505,E2 -26684.505} C_VEL
LIN {X 0,Y 122.285,Z 398.942,A -85,B 0,C 180,E1 -26686.105,E2 -26686.105} C_VEL
LIN {X 0,Y 118.943,Z 411.054,A -85,B 0,C 180,E1 -26688.332,E2 -26688.332} C_VEL
LIN {X 0,Y 116.101,Z 420.028,A -85,B 0,C 180,E1 -26690.529,E2 -26690.529} C_VEL
LIN {X 0,Y 112.65,Z 429.848,A -85,B 0,C 180,E1 -26693.646,E2 -26693.646} C_VEL
LIN {X 0,Y 108.507,Z 440.121,A -85,B 0,C 180,E1 -26697.892,E2 -26697.892} C_VEL
LIN {X 0,Y 105.956,Z 446.446,A -85,B 0,C 180,E1 -26701.25,E2 -26701.25} C_VEL
LIN {X 0,Y 102.595,Z 454.694,A -85,B 0,C 180,E1 -26706.797,E2 -26706.797} C_VEL
LIN {X 0,Y 100.5,Z 460.286,A -85,B 0,C 180,E1 -26711.652,E2 -26711.652} C_VEL
LIN {X 0,Y 98.887,Z 465.733,A -85,B 0,C 180,E1 -26717.683,E2 -26717.683} C_VEL
LIN {X 0,Y 98.078,Z 469.952,A -85,B 0,C 180,E1 -26723.823,E2 -26723.823} C_VEL
LIN {X 0,Y 98.028,Z 473.078,A -85,B 0,C 180,E1 -26729.994,E2 -26729.994} C_VEL
LIN {X 0,Y 98.015,Z 474.606,A -85,B 0,C 180,E1 -26734.105,E2 -26734.105} C_VEL
LIN {X 0,Y 98.297,Z 475.712,A -85,B 0,C 180,E1 -26738.215,E2 -26738.215} C_VEL
LIN {X 0,Y 100.138,Z 476.713,A -85,B 0,C 180,E1 -26746.297,E2 -26746.297} C_VEL
LIN {X 0,Y 103.675,Z 476.228,A -85,B 0,C 180,E1 -26753.993,E2 -26753.993} C_VEL
LIN {X 0,Y 109.145,Z 474.16,A -85,B 0,C 180,E1 -26760.999,E2 -26760.999} C_VEL
LIN {X 0,Y 116.058,Z 470.519,A -85,B 0,C 180,E1 -26767.262,E2 -26767.262} C_VEL
LIN {X 0,Y 122.454,Z 466.334,A -85,B 0,C 180,E1 -26771.729,E2 -26771.729} C_VEL
LIN {X 0,Y 128.627,Z 461.629,A -85,B 0,C 180,E1 -26775.252,E2 -26775.252} C_VEL
LIN {X 0,Y 135.828,Z 455.387,A -85,B 0,C 180,E1 -26778.605,E2 -26778.605} C_VEL
LIN {X 0,Y 143.508,Z 447.602,A -85,B 0,C 180,E1 -26781.58,E2 -26781.58} C_VEL
LIN {X 0,Y 150.15,Z 439.714,A -85,B 0,C 180,E1 -26783.836,E2 -26783.836} C_VEL
LIN {X 0,Y 156.318,Z 431.182,A -85,B 0,C 180,E1 -26785.696,E2 -26785.696} C_VEL
LIN {X 0,Y 162.737,Z 420.755,A -85,B 0,C 180,E1 -26787.358,E2 -26787.358} C_VEL
LIN {X 0,Y 168.518,Z 409.192,A -85,B 0,C 180,E1 -26788.746,E2 -26788.746} C_VEL
LIN {X 0,Y 173.059,Z 397.599,A -85,B 0,C 180,E1 -26789.751,E2 -26789.751} C_VEL
LIN {X 0,Y 175.74,Z 389.002,A -85,B 0,C 180,E1 -26790.31,E2 -26790.31} C_VEL
LIN {X 0,Y 177.276,Z 382.319,A -85,B 0,C 180,E1 -26790.798,E2 -26790.798} C_VEL
LIN {X 0,Y 177.88,Z 377.169,A -85,B 0,C 180,E1 -26791.449,E2 -26791.449} C_VEL
LIN {X 0,Y 177.834,Z 372.632,A -85,B 0,C 180,E1 -26792.4,E2 -26792.4} C_VEL
LIN {X 0,Y 177.349,Z 369.951,A -85,B 0,C 180,E1 -26793.357,E2 -26793.357} C_VEL
LIN {X 0,Y 175.493,Z 363.953,A -85,B 0,C 180,E1 -26796.542,E2 -26796.542} C_VEL
LIN {X 0,Y 174.12,Z 360.168,A -85,B 0,C 180,E1 -26799.275,E2 -26799.275} C_VEL
LIN {X 0,Y 173.39,Z 358.403,A -85,B 0,C 180,E1 -26801.07,E2 -26801.07} C_VEL
LIN {X 0,Y 172.084,Z 354.829,A -85,B 0,C 180,E1 -26806.535,E2 -26806.535} C_VEL
LIN {X 0,Y 172.251,Z 354.801,A -85,B 0,C 180,E1 -26813.528,E2 -26813.528} C_VEL
LIN {X 0,Y 172.466,Z 355.461,A -85,B 0,C 180,E1 -26814.71,E2 -26814.71} C_VEL
LIN {X 0,Y 173.874,Z 358.955,A -85,B 0,C 180,E1 -26819.267,E2 -26819.267} C_VEL
LIN {X 0,Y 175.441,Z 362.661,A -85,B 0,C 180,E1 -26822.402,E2 -26822.402} C_VEL
LIN {X 0,Y 177.036,Z 366.338,A -85,B 0,C 180,E1 -26824.966,E2 -26824.966} C_VEL
LIN {X 0,Y 177.586,Z 368.062,A -85,B 0,C 180,E1 -26825.851,E2 -26825.851} C_VEL
LIN {X 0,Y 175.121,Z 381.539,A -85,B 0,C 180,E1 -26826.377,E2 -26826.377} C_VEL
LIN {X 0,Y 171.433,Z 394.315,A -85,B 0,C 180,E1 -26827.121,E2 -26827.121} C_VEL
LIN {X 0,Y 166.808,Z 406.201,A -85,B 0,C 180,E1 -26828.096,E2 -26828.096} C_VEL
LIN {X 0,Y 161.162,Z 417.635,A -85,B 0,C 180,E1 -26829.411,E2 -26829.411} C_VEL
LIN {X 0,Y 154.812,Z 427.961,A -85,B 0,C 180,E1 -26830.998,E2 -26830.998} C_VEL
LIN {X 0,Y 147.822,Z 437.428,A -85,B 0,C 180,E1 -26832.95,E2 -26832.95} C_VEL
LIN {X 0,Y 140.27,Z 446.053,A -85,B 0,C 180,E1 -26835.359,E2 -26835.359} C_VEL
LIN {X 0,Y 133.038,Z 453.101,A -85,B 0,C 180,E1 -26838.048,E2 -26838.048} C_VEL
LIN {X 0,Y 124.764,Z 459.891,A -85,B 0,C 180,E1 -26841.665,E2 -26841.665} C_VEL
LIN {X 0,Y 117.126,Z 465.191,A -85,B 0,C 180,E1 -26845.848,E2 -26845.848} C_VEL
LIN {X 0,Y 109.974,Z 469.294,A -85,B 0,C 180,E1 -26850.729,E2 -26850.729} C_VEL
LIN {X 0,Y 104.113,Z 471.993,A -85,B 0,C 180,E1 -26855.911,E2 -26855.911} C_VEL
LIN {X 0,Y 100.617,Z 473.267,A -85,B 0,C 180,E1 -26859.805,E2 -26859.805} C_VEL
LIN {X 0,Y 95.661,Z 474.296,A -85,B 0,C 180,E1 -26867.254,E2 -26867.254} C_VEL
LIN {X 0,Y 93.097,Z 474.199,A -85,B 0,C 180,E1 -26872.857,E2 -26872.857} C_VEL
LIN {X 0,Y 91.636,Z 473.563,A -85,B 0,C 180,E1 -26877.538,E2 -26877.538} C_VEL
LIN {X 0,Y 90.681,Z 472.496,A -85,B 0,C 180,E1 -26882.297,E2 -26882.297} C_VEL
LIN {X 0,Y 90.24,Z 470.171,A -85,B 0,C 180,E1 -26889.105,E2 -26889.105} C_VEL
LIN {X 0,Y 90.868,Z 466.449,A -85,B 0,C 180,E1 -26896.591,E2 -26896.591} C_VEL
LIN {X 0,Y 92.518,Z 461.141,A -85,B 0,C 180,E1 -26904.176,E2 -26904.176} C_VEL
LIN {X 0,Y 94.966,Z 454.579,A -85,B 0,C 180,E1 -26911.067,E2 -26911.067} C_VEL
LIN {X 0,Y 98.227,Z 446.821,A -85,B 0,C 180,E1 -26917.199,E2 -26917.199} C_VEL
LIN {X 0,Y 101.853,Z 438.828,A -85,B 0,C 180,E1 -26921.953,E2 -26921.953} C_VEL
LIN {X 0,Y 105.913,Z 429.052,A -85,B 0,C 180,E1 -26926.386,E2 -26926.386} C_VEL
LIN {X 0,Y 110.107,Z 418.149,A -85,B 0,C 180,E1 -26930.07,E2 -26930.07} C_VEL
LIN {X 0,Y 113.99,Z 406.329,A -85,B 0,C 180,E1 -26933.023,E2 -26933.023} C_VEL
LIN {X 0,Y 117.262,Z 393.898,A -85,B 0,C 180,E1 -26935.269,E2 -26935.269} C_VEL
LIN {X 0,Y 119.899,Z 380.682,A -85,B 0,C 180,E1 -26936.931,E2 -26936.931} C_VEL
LIN {X 0,Y 121.696,Z 367.22,A -85,B 0,C 180,E1 -26937.946,E2 -26937.946} C_VEL
LIN {X 0,Y 124.873,Z 326.626,A -85,B 0,C 180,E1 -26939.915,E2 -26939.915} C_VEL
LIN {X 0,Y 122.274,Z 319.867,A -85,B 0,C 180,E1 -26941.596,E2 -26941.596} C_VEL
LIN {X 0,Y 117.387,Z 310.1,A -85,B 0,C 180,E1 -26944.816,E2 -26944.816} C_VEL
LIN {X 0,Y 113.3,Z 302.855,A -85,B 0,C 180,E1 -26947.801,E2 -26947.801} C_VEL
LIN {X 0,Y 109.523,Z 296.915,A -85,B 0,C 180,E1 -26950.86,E2 -26950.86} C_VEL
LIN {X 0,Y 107.358,Z 293.802,A -85,B 0,C 180,E1 -26952.785,E2 -26952.785} C_VEL
LIN {X 0,Y 105.202,Z 290.659,A -85,B 0,C 180,E1 -26954.856,E2 -26954.856} C_VEL
LIN {X 0,Y 102.65,Z 287.372,A -85,B 0,C 180,E1 -26957.527,E2 -26957.527} C_VEL
LIN {X 0,Y 101.944,Z 286.143,A -85,B 0,C 180,E1 -26958.375,E2 -26958.375} C_VEL
LIN {X 0,Y 99.466,Z 283.664,A -85,B 0,C 180,E1 -26961.349,E2 -26961.349} C_VEL
LIN {X 0,Y 98.244,Z 281.181,A -85,B 0,C 180,E1 -26963.215,E2 -26963.215} C_VEL
LIN {X 0,Y 95.468,Z 279.246,A -85,B 0,C 180,E1 -26967.369,E2 -26967.369} C_VEL
LIN {X 0,Y 93.968,Z 276.902,A -85,B 0,C 180,E1 -26970.472,E2 -26970.472} C_VEL
LIN {X 0,Y 93.632,Z 275.82,A -85,B 0,C 180,E1 -26972.043,E2 -26972.043} C_VEL
LIN {X 0,Y 93.626,Z 275.366,A -85,B 0,C 180,E1 -26974.274,E2 -26974.274} C_VEL
LIN {X 0,Y 93.644,Z 275.294,A -85,B 0,C 180,E1 -26977.979,E2 -26977.979} C_VEL
LIN {X 0,Y 94.019,Z 275.226,A -85,B 0,C 180,E1 -26987.059,E2 -26987.059} C_VEL
LIN {X 0,Y 94.16,Z 275.231,A -85,B 0,C 180,E1 -26991.432,E2 -26991.432} C_VEL
LIN {X 0,Y 94.749,Z 275.129,A -85,B 0,C 180,E1 -27000.016,E2 -27000.016} C_VEL
LIN {X 0,Y 94.24,Z 275.579,A -85,B 0,C 180,E1 -27007.515,E2 -27007.515} C_VEL
LIN {X 0,Y 94.448,Z 276.617,A -85,B 0,C 180,E1 -27009.114,E2 -27009.114} C_VEL
LIN {X 0,Y 95.802,Z 279.037,A -85,B 0,C 180,E1 -27011.923,E2 -27011.923} C_VEL
LIN {X 0,Y 98.49,Z 281.312,A -85,B 0,C 180,E1 -27015.935,E2 -27015.935} C_VEL
LIN {X 0,Y 100.396,Z 284.594,A -85,B 0,C 180,E1 -27018.642,E2 -27018.642} C_VEL
LIN {X 0,Y 102.44,Z 286.613,A -85,B 0,C 180,E1 -27020.995,E2 -27020.995} C_VEL
LIN {X 0,Y 104.718,Z 290.09,A -85,B 0,C 180,E1 -27023.499,E2 -27023.499} C_VEL
LIN {X 0,Y 106.112,Z 291.749,A -85,B 0,C 180,E1 -27024.844,E2 -27024.844} C_VEL
LIN {X 0,Y 109.217,Z 296.381,A -85,B 0,C 180,E1 -27027.694,E2 -27027.694} C_VEL
LIN {X 0,Y 113.924,Z 303.968,A -85,B 0,C 180,E1 -27031.511,E2 -27031.511} C_VEL
LIN {X 0,Y 118.632,Z 312.539,A -85,B 0,C 180,E1 -27034.873,E2 -27034.873} C_VEL
LIN {X 0,Y 120.66,Z 317.058,A -85,B 0,C 180,E1 -27036.254,E2 -27036.254} C_VEL
LIN {X 0,Y 123.967,Z 327.432,A -85,B 0,C 180,E1 -27038.595,E2 -27038.595} C_VEL
LIN {X 0,Y 124.736,Z 330.081,A -85,B 0,C 180,E1 -27039.132,E2 -27039.132} C_VEL
LIN {X 0,Y 121.264,Z 373.263,A -85,B 0,C 180,E1 -27041.262,E2 -27041.262} C_VEL
LIN {X 0,Y 119.244,Z 386.287,A -85,B 0,C 180,E1 -27042.383,E2 -27042.383} C_VEL
LIN {X 0,Y 116.681,Z 398.447,A -85,B 0,C 180,E1 -27044.019,E2 -27044.019} C_VEL
LIN {X 0,Y 113.178,Z 410.676,A -85,B 0,C 180,E1 -27046.297,E2 -27046.297} C_VEL
LIN {X 0,Y 110.161,Z 419.691,A -85,B 0,C 180,E1 -27048.548,E2 -27048.548} C_VEL
LIN {X 0,Y 106.505,Z 429.557,A -85,B 0,C 180,E1 -27051.776,E2 -27051.776} C_VEL
LIN {X 0,Y 102.63,Z 438.486,A -85,B 0,C 180,E1 -27055.509,E2 -27055.509} C_VEL
LIN {X 0,Y 99.767,Z 445.465,A -85,B 0,C 180,E1 -27059.281,E2 -27059.281} C_VEL
LIN {X 0,Y 96.094,Z 453.864,A -85,B 0,C 180,E1 -27065.125,E2 -27065.125} C_VEL
LIN {X 0,Y 93.373,Z 460.606,A -85,B 0,C 180,E1 -27071.337,E2 -27071.337} C_VEL
LIN {X 0,Y 91.533,Z 466.744,A -85,B 0,C 180,E1 -27078.926,E2 -27078.926} C_VEL
LIN {X 0,Y 90.905,Z 470.694,A -85,B 0,C 180,E1 -27085.559,E2 -27085.559} C_VEL
LIN {X 0,Y 90.955,Z 472.71,A -85,B 0,C 180,E1 -27089.993,E2 -27089.993} C_VEL
LIN {X 0,Y 90.934,Z 474.284,A -85,B 0,C 180,E1 -27094.426,E2 -27094.426} C_VEL
LIN {X 0,Y 91.269,Z 475.46,A -85,B 0,C 180,E1 -27098.852,E2 -27098.852} C_VEL
LIN {X 0,Y 92.095,Z 476.225,A -85,B 0,C 180,E1 -27103.227,E2 -27103.227} C_VEL
LIN {X 0,Y 95.064,Z 476.582,A -85,B 0,C 180,E1 -27111.686,E2 -27111.686} C_VEL
LIN {X 0,Y 97.21,Z 476.206,A -85,B 0,C 180,E1 -27115.7,E2 -27115.7} C_VEL
LIN {X 0,Y 99.948,Z 475.458,A -85,B 0,C 180,E1 -27119.479,E2 -27119.479} C_VEL
LIN {X 0,Y 106.608,Z 472.724,A -85,B 0,C 180,E1 -27126.385,E2 -27126.385} C_VEL
LIN {X 0,Y 112.581,Z 469.603,A -85,B 0,C 180,E1 -27130.948,E2 -27130.948} C_VEL
LIN {X 0,Y 119.045,Z 465.475,A -85,B 0,C 180,E1 -27135.1,E2 -27135.1} C_VEL
LIN {X 0,Y 127.447,Z 459.211,A -85,B 0,C 180,E1 -27139.301,E2 -27139.301} C_VEL
LIN {X 0,Y 135.232,Z 452.408,A -85,B 0,C 180,E1 -27142.415,E2 -27142.415} C_VEL
LIN {X 0,Y 143.297,Z 443.963,A -85,B 0,C 180,E1 -27145.227,E2 -27145.227} C_VEL
LIN {X 0,Y 150.303,Z 435.348,A -85,B 0,C 180,E1 -27147.307,E2 -27147.307} C_VEL
LIN {X 0,Y 157.603,Z 424.75,A -85,B 0,C 180,E1 -27149.13,E2 -27149.13} C_VEL
LIN {X 0,Y 163.51,Z 414.253,A -85,B 0,C 180,E1 -27150.495,E2 -27150.495} C_VEL
LIN {X 0,Y 168.967,Z 402.044,A -85,B 0,C 180,E1 -27151.644,E2 -27151.644} C_VEL
LIN {X 0,Y 173.29,Z 389.357,A -85,B 0,C 180,E1 -27152.49,E2 -27152.49} C_VEL
LIN {X 0,Y 176.39,Z 376.438,A -85,B 0,C 180,E1 -27153.05,E2 -27153.05} C_VEL
LIN {X 0,Y 177.395,Z 370.098,A -85,B 0,C 180,E1 -27153.285,E2 -27153.285} C_VEL
LIN {X 0,Y 177.349,Z 369.951,A -85,B 0,C 180,E1 -27153.357,E2 -27153.357} C_VEL
LIN {X 0,Y 176.611,Z 368.152,A -85,B 0,C 180,E1 -27154.463,E2 -27154.463} C_VEL
LIN {X 0,Y 175.351,Z 366.563,A -85,B 0,C 180,E1 -27156.278,E2 -27156.278} C_VEL
LIN {X 0,Y 173.309,Z 365.617,A -85,B 0,C 180,E1 -27159.504,E2 -27159.504} C_VEL
LIN {X 0,Y 172.062,Z 364.945,A -85,B 0,C 180,E1 -27162.172,E2 -27162.172} C_VEL
LIN {X 0,Y 171.659,Z 364.177,A -85,B 0,C 180,E1 -27163.498,E2 -27163.498} C_VEL
LIN {X 0,Y 171.114,Z 361.834,A -85,B 0,C 180,E1 -27166.936,E2 -27166.936} C_VEL
LIN {X 0,Y 171.334,Z 361.85,A -85,B 0,C 180,E1 -27173.493,E2 -27173.493} C_VEL
LIN {X 0,Y 172.669,Z 365.775,A -85,B 0,C 180,E1 -27178.679,E2 -27178.679} C_VEL
LIN {X 0,Y 173.901,Z 369.126,A -85,B 0,C 180,E1 -27181.583,E2 -27181.583} C_VEL
LIN {X 0,Y 175.021,Z 372.188,A -85,B 0,C 180,E1 -27183.797,E2 -27183.797} C_VEL
LIN {X 0,Y 172.221,Z 384.921,A -85,B 0,C 180,E1 -27184.296,E2 -27184.296} C_VEL
LIN {X 0,Y 168.005,Z 398.068,A -85,B 0,C 180,E1 -27185.095,E2 -27185.095} C_VEL
LIN {X 0,Y 163.404,Z 408.807,A -85,B 0,C 180,E1 -27185.996,E2 -27185.996} C_VEL
LIN {X 0,Y 157.623,Z 419.656,A -85,B 0,C 180,E1 -27187.257,E2 -27187.257} C_VEL
LIN {X 0,Y 151.036,Z 429.768,A -85,B 0,C 180,E1 -27188.82,E2 -27188.82} C_VEL
LIN {X 0,Y 144.706,Z 437.895,A -85,B 0,C 180,E1 -27190.454,E2 -27190.454} C_VEL
LIN {X 0,Y 136.903,Z 446.435,A -85,B 0,C 180,E1 -27192.764,E2 -27192.764} C_VEL
LIN {X 0,Y 129.026,Z 453.717,A -85,B 0,C 180,E1 -27195.509,E2 -27195.509} C_VEL
LIN {X 0,Y 122.11,Z 459.145,A -85,B 0,C 180,E1 -27198.276,E2 -27198.276} C_VEL
LIN {X 0,Y 113.933,Z 464.632,A -85,B 0,C 180,E1 -27202.305,E2 -27202.305} C_VEL
LIN {X 0,Y 105.082,Z 469.444,A -85,B 0,C 180,E1 -27207.897,E2 -27207.897} C_VEL
LIN {X 0,Y 99.716,Z 471.76,A -85,B 0,C 180,E1 -27212.259,E2 -27212.259} C_VEL
LIN {X 0,Y 95.8,Z 473.121,A -85,B 0,C 180,E1 -27216.21,E2 -27216.21} C_VEL
LIN {X 0,Y 92.339,Z 474.015,A -85,B 0,C 180,E1 -27220.449,E2 -27220.449} C_VEL
LIN {X 0,Y 89.423,Z 474.402,A -85,B 0,C 180,E1 -27224.992,E2 -27224.992} C_VEL
LIN {X 0,Y 87.011,Z 474.356,A -85,B 0,C 180,E1 -27229.756,E2 -27229.756} C_VEL
LIN {X 0,Y 84.861,Z 473.656,A -85,B 0,C 180,E1 -27235.876,E2 -27235.876} C_VEL
LIN {X 0,Y 83.262,Z 471.433,A -85,B 0,C 180,E1 -27245.045,E2 -27245.045} C_VEL
LIN {X 0,Y 83.32,Z 468.386,A -85,B 0,C 180,E1 -27252.837,E2 -27252.837} C_VEL
LIN {X 0,Y 84.393,Z 464.227,A -85,B 0,C 180,E1 -27260.42,E2 -27260.42} C_VEL
LIN {X 0,Y 86.361,Z 458.851,A -85,B 0,C 180,E1 -27267.675,E2 -27267.675} C_VEL
LIN {X 0,Y 89.248,Z 452.074,A -85,B 0,C 180,E1 -27274.524,E2 -27274.524} C_VEL
LIN {X 0,Y 92.846,Z 444.403,A -85,B 0,C 180,E1 -27280.357,E2 -27280.357} C_VEL
LIN {X 0,Y 97.179,Z 434.976,A -85,B 0,C 180,E1 -27285.742,E2 -27285.742} C_VEL
LIN {X 0,Y 101.821,Z 424.211,A -85,B 0,C 180,E1 -27290.195,E2 -27290.195} C_VEL
LIN {X 0,Y 105.888,Z 413.523,A -85,B 0,C 180,E1 -27293.474,E2 -27293.474} C_VEL
LIN {X 0,Y 109.797,Z 401.32,A -85,B 0,C 180,E1 -27296.215,E2 -27296.215} C_VEL
LIN {X 0,Y 113.066,Z 388.129,A -85,B 0,C 180,E1 -27298.297,E2 -27298.297} C_VEL
LIN {X 0,Y 115.436,Z 375.039,A -85,B 0,C 180,E1 -27299.661,E2 -27299.661} C_VEL
LIN {X 0,Y 117.094,Z 358.696,A -85,B 0,C 180,E1 -27300.638,E2 -27300.638} C_VEL
LIN {X 0,Y 119.561,Z 328.448,A -85,B 0,C 180,E1 -27302.108,E2 -27302.108} C_VEL
LIN {X 0,Y 115.834,Z 319.722,A -85,B 0,C 180,E1 -27304.74,E2 -27304.74} C_VEL
LIN {X 0,Y 111.039,Z 310.343,A -85,B 0,C 180,E1 -27308.418,E2 -27308.418} C_VEL
LIN {X 0,Y 106.361,Z 302.47,A -85,B 0,C 180,E1 -27312.504,E2 -27312.504} C_VEL
LIN {X 0,Y 102.278,Z 296.415,A -85,B 0,C 180,E1 -27316.618,E2 -27316.618} C_VEL
LIN {X 0,Y 99.774,Z 292.748,A -85,B 0,C 180,E1 -27319.58,E2 -27319.58} C_VEL
LIN {X 0,Y 96.83,Z 289.163,A -85,B 0,C 180,E1 -27323.562,E2 -27323.562} C_VEL
LIN {X 0,Y 96.162,Z 287.758,A -85,B 0,C 180,E1 -27324.692,E2 -27324.692} C_VEL
LIN {X 0,Y 93.091,Z 284.987,A -85,B 0,C 180,E1 -27330.01,E2 -27330.01} C_VEL
LIN {X 0,Y 91.784,Z 282.387,A -85,B 0,C 180,E1 -27333.342,E2 -27333.342} C_VEL
LIN {X 0,Y 88.647,Z 279.844,A -85,B 0,C 180,E1 -27348.587,E2 -27348.587} C_VEL
LIN {X 0,Y 89.752,Z 280.338,A -85,B 0,C 180,E1 -27358.896,E2 -27358.896} C_VEL
LIN {X 0,Y 92.459,Z 282.456,A -85,B 0,C 180,E1 -27366.947,E2 -27366.947} C_VEL
LIN {X 0,Y 93.862,Z 285.313,A -85,B 0,C 180,E1 -27370.231,E2 -27370.231} C_VEL
LIN {X 0,Y 96.435,Z 287.877,A -85,B 0,C 180,E1 -27374.524,E2 -27374.524} C_VEL
LIN {X 0,Y 98.601,Z 291.34,A -85,B 0,C 180,E1 -27377.75,E2 -27377.75} C_VEL
LIN {X 0,Y 100.032,Z 292.964,A -85,B 0,C 180,E1 -27379.544,E2 -27379.544} C_VEL
LIN {X 0,Y 102.677,Z 296.739,A -85,B 0,C 180,E1 -27382.611,E2 -27382.611} C_VEL
LIN {X 0,Y 106.369,Z 302.436,A -85,B 0,C 180,E1 -27386.329,E2 -27386.329} C_VEL
LIN {X 0,Y 111.06,Z 310.375,A -85,B 0,C 180,E1 -27390.429,E2 -27390.429} C_VEL
LIN {X 0,Y 115.704,Z 319.601,A -85,B 0,C 180,E1 -27394.01,E2 -27394.01} C_VEL
LIN {X 0,Y 118.482,Z 328.497,A -85,B 0,C 180,E1 -27396.214,E2 -27396.214} C_VEL
LIN {X 0,Y 119.413,Z 331.779,A -85,B 0,C 180,E1 -27396.938,E2 -27396.938} C_VEL
LIN {X 0,Y 115.886,Z 373.349,A -85,B 0,C 180,E1 -27399.034,E2 -27399.034} C_VEL
LIN {X 0,Y 113.657,Z 386.958,A -85,B 0,C 180,E1 -27400.242,E2 -27400.242} C_VEL
LIN {X 0,Y 110.969,Z 398.907,A -85,B 0,C 180,E1 -27401.905,E2 -27401.905} C_VEL
LIN {X 0,Y 107.575,Z 410.174,A -85,B 0,C 180,E1 -27404.05,E2 -27404.05} C_VEL
LIN {X 0,Y 104.373,Z 419.24,A -85,B 0,C 180,E1 -27406.347,E2 -27406.347} C_VEL
LIN {X 0,Y 100.474,Z 429.176,A -85,B 0,C 180,E1 -27409.675,E2 -27409.675} C_VEL
LIN {X 0,Y 96.851,Z 437.254,A -85,B 0,C 180,E1 -27413.125,E2 -27413.125} C_VEL
LIN {X 0,Y 93.716,Z 444.359,A -85,B 0,C 180,E1 -27417.057,E2 -27417.057} C_VEL
LIN {X 0,Y 90.268,Z 451.68,A -85,B 0,C 180,E1 -27422.143,E2 -27422.143} C_VEL
LIN {X 0,Y 87.036,Z 458.843,A -85,B 0,C 180,E1 -27428.685,E2 -27428.685} C_VEL
LIN {X 0,Y 85.009,Z 464.541,A -85,B 0,C 180,E1 -27435.632,E2 -27435.632} C_VEL
LIN {X 0,Y 83.973,Z 468.991,A -85,B 0,C 180,E1 -27442.781,E2 -27442.781} C_VEL
LIN {X 0,Y 83.852,Z 472.329,A -85,B 0,C 180,E1 -27449.993,E2 -27449.993} C_VEL
LIN {X 0,Y 83.874,Z 473.957,A -85,B 0,C 180,E1 -27454.799,E2 -27454.799} C_VEL
LIN {X 0,Y 85.2,Z 476.029,A -85,B 0,C 180,E1 -27464.32,E2 -27464.32} C_VEL
LIN {X 0,Y 88.47,Z 476.508,A -85,B 0,C 180,E1 -27473.395,E2 -27473.395} C_VEL
LIN {X 0,Y 93.821,Z 475.489,A -85,B 0,C 180,E1 -27481.617,E2 -27481.617} C_VEL
LIN {X 0,Y 97.243,Z 474.413,A -85,B 0,C 180,E1 -27485.315,E2 -27485.315} C_VEL
LIN {X 0,Y 100.974,Z 472.907,A -85,B 0,C 180,E1 -27488.778,E2 -27488.778} C_VEL
LIN {X 0,Y 109.541,Z 468.663,A -85,B 0,C 180,E1 -27494.881,E2 -27494.881} C_VEL
LIN {X 0,Y 116.617,Z 464.283,A -85,B 0,C 180,E1 -27498.87,E2 -27498.87} C_VEL
LIN {X 0,Y 124.265,Z 458.763,A -85,B 0,C 180,E1 -27502.345,E2 -27502.345} C_VEL
LIN {X 0,Y 132.414,Z 451.893,A -85,B 0,C 180,E1 -27505.345,E2 -27505.345} C_VEL
LIN {X 0,Y 140.839,Z 443.344,A -85,B 0,C 180,E1 -27508.02,E2 -27508.02} C_VEL
LIN {X 0,Y 148.128,Z 434.616,A -85,B 0,C 180,E1 -27509.974,E2 -27509.974} C_VEL
LIN {X 0,Y 155.647,Z 423.889,A -85,B 0,C 180,E1 -27511.692,E2 -27511.692} C_VEL
LIN {X 0,Y 161.712,Z 413.153,A -85,B 0,C 180,E1 -27512.981,E2 -27512.981} C_VEL
LIN {X 0,Y 167.031,Z 401.351,A -85,B 0,C 180,E1 -27514.015,E2 -27514.015} C_VEL
LIN {X 0,Y 170.983,Z 390.043,A -85,B 0,C 180,E1 -27514.717,E2 -27514.717} C_VEL
LIN {X 0,Y 174.159,Z 377.589,A -85,B 0,C 180,E1 -27515.234,E2 -27515.234} C_VEL
LIN {X 0,Y 174.775,Z 373.907,A -85,B 0,C 180,E1 -27515.421,E2 -27515.421} C_VEL
LIN {X 0,Y 173.618,Z 369.446,A -85,B 0,C 180,E1 -27518.035,E2 -27518.035} C_VEL
LIN {X 0,Y 172.732,Z 366.565,A -85,B 0,C 180,E1 -27520.226,E2 -27520.226} C_VEL
LIN {X 0,Y 172.174,Z 365.132,A -85,B 0,C 180,E1 -27521.827,E2 -27521.827} C_VEL
LIN {X 0,Y 171.659,Z 364.177,A -85,B 0,C 180,E1 -27523.498,E2 -27523.498} C_VEL
LIN {X 0,Y 171.188,Z 363.5,A -85,B 0,C 180,E1 -27525.453,E2 -27525.453} C_VEL
LIN {X 0,Y 170.64,Z 364.42,A -85,B 0,C 180,E1 -27528.089,E2 -27528.089} C_VEL
LIN {X 0,Y 170.382,Z 369.463,A -85,B 0,C 180,E1 -27534.016,E2 -27534.016} C_VEL
LIN {X 0,Y 171.306,Z 372.635,A -85,B 0,C 180,E1 -27538.228,E2 -27538.228} C_VEL
LIN {X 0,Y 172.459,Z 376.567,A -85,B 0,C 180,E1 -27541.619,E2 -27541.619} C_VEL
LIN {X 0,Y 169.223,Z 389.165,A -85,B 0,C 180,E1 -27542.2,E2 -27542.2} C_VEL
LIN {X 0,Y 165.174,Z 400.49,A -85,B 0,C 180,E1 -27542.9,E2 -27542.9} C_VEL
LIN {X 0,Y 160.228,Z 411.259,A -85,B 0,C 180,E1 -27543.807,E2 -27543.807} C_VEL
LIN {X 0,Y 153.7,Z 422.648,A -85,B 0,C 180,E1 -27545.133,E2 -27545.133} C_VEL
LIN {X 0,Y 145.982,Z 433.419,A -85,B 0,C 180,E1 -27546.85,E2 -27546.85} C_VEL
LIN {X 0,Y 138.477,Z 442.112,A -85,B 0,C 180,E1 -27548.746,E2 -27548.746} C_VEL
LIN {X 0,Y 130.648,Z 449.749,A -85,B 0,C 180,E1 -27550.998,E2 -27550.998} C_VEL
LIN {X 0,Y 121.406,Z 457.286,A -85,B 0,C 180,E1 -27554.18,E2 -27554.18} C_VEL
LIN {X 0,Y 111.825,Z 463.69,A -85,B 0,C 180,E1 -27558.3,E2 -27558.3} C_VEL
LIN {X 0,Y 103.121,Z 468.412,A -85,B 0,C 180,E1 -27563.081,E2 -27563.081} C_VEL
LIN {X 0,Y 95.76,Z 471.532,A -85,B 0,C 180,E1 -27568.288,E2 -27568.288} C_VEL
LIN {X 0,Y 90.843,Z 473.12,A -85,B 0,C 180,E1 -27572.767,E2 -27572.767} C_VEL
LIN {X 0,Y 87.456,Z 473.956,A -85,B 0,C 180,E1 -27576.537,E2 -27576.537} C_VEL
LIN {X 0,Y 83.31,Z 474.51,A -85,B 0,C 180,E1 -27582.417,E2 -27582.417} C_VEL
LIN {X 0,Y 78.98,Z 474.097,A -85,B 0,C 180,E1 -27591.483,E2 -27591.483} C_VEL
LIN {X 0,Y 77.355,Z 473.227,A -85,B 0,C 180,E1 -27596.977,E2 -27596.977} C_VEL
LIN {X 0,Y 76.066,Z 470.368,A -85,B 0,C 180,E1 -27607.45,E2 -27607.45} C_VEL
LIN {X 0,Y 76.633,Z 466.448,A -85,B 0,C 180,E1 -27616.754,E2 -27616.754} C_VEL
LIN {X 0,Y 78.273,Z 461.657,A -85,B 0,C 180,E1 -27624.857,E2 -27624.857} C_VEL
LIN {X 0,Y 80.791,Z 455.577,A -85,B 0,C 180,E1 -27632.501,E2 -27632.501} C_VEL
LIN {X 0,Y 84.473,Z 447.974,A -85,B 0,C 180,E1 -27639.586,E2 -27639.586} C_VEL
LIN {X 0,Y 88.523,Z 440.172,A -85,B 0,C 180,E1 -27644.96,E2 -27644.96} C_VEL
LIN {X 0,Y 93.028,Z 430.737,A -85,B 0,C 180,E1 -27649.882,E2 -27649.882} C_VEL
LIN {X 0,Y 97.67,Z 420.146,A -85,B 0,C 180,E1 -27653.883,E2 -27653.883} C_VEL
LIN {X 0,Y 102.133,Z 408.223,A -85,B 0,C 180,E1 -27657.185,E2 -27657.185} C_VEL
LIN {X 0,Y 105.836,Z 396.001,A -85,B 0,C 180,E1 -27659.603,E2 -27659.603} C_VEL
LIN {X 0,Y 108.906,Z 382.561,A -85,B 0,C 180,E1 -27661.43,E2 -27661.43} C_VEL
LIN {X 0,Y 110.927,Z 369.811,A -85,B 0,C 180,E1 -27662.522,E2 -27662.522} C_VEL
LIN {X 0,Y 114.405,Z 330.547,A -85,B 0,C 180,E1 -27664.483,E2 -27664.483} C_VEL
LIN {X 0,Y 110.471,Z 321.464,A -85,B 0,C 180,E1 -27667.617,E2 -27667.617} C_VEL
LIN {X 0,Y 106.895,Z 314.401,A -85,B 0,C 180,E1 -27670.726,E2 -27670.726} C_VEL
LIN {X 0,Y 102.405,Z 306.482,A -85,B 0,C 180,E1 -27675.157,E2 -27675.157} C_VEL
LIN {X 0,Y 99.553,Z 302.271,A -85,B 0,C 180,E1 -27678.372,E2 -27678.372} C_VEL
LIN {X 0,Y 96.795,Z 298.205,A -85,B 0,C 180,E1 -27682.012,E2 -27682.012} C_VEL
LIN {X 0,Y 94.5,Z 294.929,A -85,B 0,C 180,E1 -27685.592,E2 -27685.592} C_VEL
LIN {X 0,Y 93.94,Z 294.116,A -85,B 0,C 180,E1 -27686.57,E2 -27686.57} C_VEL
LIN {X 0,Y 91.231,Z 291.078,A -85,B 0,C 180,E1 -27692.023,E2 -27692.023} C_VEL
LIN {X 0,Y 90.475,Z 289.223,A -85,B 0,C 180,E1 -27694.282,E2 -27694.282} C_VEL
LIN {X 0,Y 87.738,Z 286.879,A -85,B 0,C 180,E1 -27708.876,E2 -27708.876} C_VEL
LIN {X 0,Y 88.83,Z 287.387,A -85,B 0,C 180,E1 -27718.884,E2 -27718.884} C_VEL
LIN {X 0,Y 90.955,Z 289.28,A -85,B 0,C 180,E1 -27725.679,E2 -27725.679} C_VEL
LIN {X 0,Y 92.473,Z 292.238,A -85,B 0,C 180,E1 -27729.471,E2 -27729.471} C_VEL
LIN {X 0,Y 94.493,Z 294.515,A -85,B 0,C 180,E1 -27733.148,E2 -27733.148} C_VEL
LIN {X 0,Y 96.7,Z 297.887,A -85,B 0,C 180,E1 -27736.645,E2 -27736.645} C_VEL
LIN {X 0,Y 97.777,Z 299.405,A -85,B 0,C 180,E1 -27738.141,E2 -27738.141} C_VEL
LIN {X 0,Y 101.005,Z 304.269,A -85,B 0,C 180,E1 -27742.129,E2 -27742.129} C_VEL
LIN {X 0,Y 104.523,Z 310.095,A -85,B 0,C 180,E1 -27745.847,E2 -27745.847} C_VEL
LIN {X 0,Y 108.976,Z 318.407,A -85,B 0,C 180,E1 -27749.952,E2 -27749.952} C_VEL
LIN {X 0,Y 111.795,Z 324.859,A -85,B 0,C 180,E1 -27752.348,E2 -27752.348} C_VEL
LIN {X 0,Y 114.279,Z 333.637,A -85,B 0,C 180,E1 -27754.57,E2 -27754.57} C_VEL
LIN {X 0,Y 110.733,Z 373.21,A -85,B 0,C 180,E1 -27756.578,E2 -27756.578} C_VEL
LIN {X 0,Y 108.468,Z 386.483,A -85,B 0,C 180,E1 -27757.751,E2 -27757.751} C_VEL
LIN {X 0,Y 105.424,Z 399.346,A -85,B 0,C 180,E1 -27759.565,E2 -27759.565} C_VEL
LIN {X 0,Y 101.54,Z 411.249,A -85,B 0,C 180,E1 -27761.914,E2 -27761.914} C_VEL
LIN {X 0,Y 98.264,Z 420.151,A -85,B 0,C 180,E1 -27764.33,E2 -27764.33} C_VEL
LIN {X 0,Y 94.155,Z 429.894,A -85,B 0,C 180,E1 -27767.786,E2 -27767.786} C_VEL
LIN {X 0,Y 89.388,Z 439.78,A -85,B 0,C 180,E1 -27772.45,E2 -27772.45} C_VEL
LIN {X 0,Y 85.409,Z 447.897,A -85,B 0,C 180,E1 -27777.657,E2 -27777.657} C_VEL
LIN {X 0,Y 82.057,Z 454.592,A -85,B 0,C 180,E1 -27783.271,E2 -27783.271} C_VEL
LIN {X 0,Y 79.554,Z 460.151,A -85,B 0,C 180,E1 -27789.298,E2 -27789.298} C_VEL
LIN {X 0,Y 77.607,Z 465.56,A -85,B 0,C 180,E1 -27796.907,E2 -27796.907} C_VEL
LIN {X 0,Y 76.766,Z 469.745,A -85,B 0,C 180,E1 -27804.739,E2 -27804.739} C_VEL
LIN {X 0,Y 76.769,Z 471.943,A -85,B 0,C 180,E1 -27809.992,E2 -27809.992} C_VEL
LIN {X 0,Y 76.801,Z 473.629,A -85,B 0,C 180,E1 -27815.242,E2 -27815.242} C_VEL
LIN {X 0,Y 78.316,Z 475.804,A -85,B 0,C 180,E1 -27825.609,E2 -27825.609} C_VEL
LIN {X 0,Y 79.856,Z 476.322,A -85,B 0,C 180,E1 -27830.603,E2 -27830.603} C_VEL
LIN {X 0,Y 84.61,Z 476.16,A -85,B 0,C 180,E1 -27839.884,E2 -27839.884} C_VEL
LIN {X 0,Y 91.522,Z 474.498,A -85,B 0,C 180,E1 -27847.894,E2 -27847.894} C_VEL
LIN {X 0,Y 95.541,Z 473.09,A -85,B 0,C 180,E1 -27851.446,E2 -27851.446} C_VEL
LIN {X 0,Y 102.287,Z 470.18,A -85,B 0,C 180,E1 -27856.164,E2 -27856.164} C_VEL
LIN {X 0,Y 109.514,Z 466.281,A -85,B 0,C 180,E1 -27860.353,E2 -27860.353} C_VEL
LIN {X 0,Y 117.355,Z 461.292,A -85,B 0,C 180,E1 -27863.937,E2 -27863.937} C_VEL
LIN {X 0,Y 125.659,Z 455.054,A -85,B 0,C 180,E1 -27867.018,E2 -27867.018} C_VEL
LIN {X 0,Y 134.314,Z 447.28,A -85,B 0,C 180,E1 -27869.686,E2 -27869.686} C_VEL
LIN {X 0,Y 143.213,Z 437.651,A -85,B 0,C 180,E1 -27872.036,E2 -27872.036} C_VEL
LIN {X 0,Y 150.907,Z 427.655,A -85,B 0,C 180,E1 -27873.692,E2 -27873.692} C_VEL
LIN {X 0,Y 157.877,Z 416.426,A -85,B 0,C 180,E1 -27875.084,E2 -27875.084} C_VEL
LIN {X 0,Y 163.736,Z 404.66,A -85,B 0,C 180,E1 -27876.139,E2 -27876.139} C_VEL
LIN {X 0,Y 168.117,Z 393.332,A -85,B 0,C 180,E1 -27876.871,E2 -27876.871} C_VEL
LIN {X 0,Y 171.9,Z 379.802,A -85,B 0,C 180,E1 -27877.441,E2 -27877.441} C_VEL
LIN {X 0,Y 172.301,Z 377.947,A -85,B 0,C 180,E1 -27877.531,E2 -27877.531} C_VEL
LIN {X 0,Y 171.367,Z 373.452,A -85,B 0,C 180,E1 -27880.647,E2 -27880.647} C_VEL
LIN {X 0,Y 170.843,Z 371.819,A -85,B 0,C 180,E1 -27882.582,E2 -27882.582} C_VEL
LIN {X 0,Y 170.07,Z 368.819,A -85,B 0,C 180,E1 -27887.461,E2 -27887.461} C_VEL
LIN {X 0,Y 170.314,Z 368.858,A -85,B 0,C 180,E1 -27893.311,E2 -27893.311} C_VEL
LIN {X 0,Y 170.382,Z 369.463,A -85,B 0,C 180,E1 -27894.016,E2 -27894.016} C_VEL
LIN {X 0,Y 170.49,Z 370.871,A -85,B 0,C 180,E1 -27895.213,E2 -27895.213} C_VEL
LIN {X 0,Y 170.365,Z 374.291,A -85,B 0,C 180,E1 -27896.779,E2 -27896.779} C_VEL
LIN {X 0,Y 169.891,Z 378.713,A -85,B 0,C 180,E1 -27898.049,E2 -27898.049} C_VEL
LIN {X 0,Y 169.01,Z 383.861,A -85,B 0,C 180,E1 -27899.055,E2 -27899.055} C_VEL
LIN {X 0,Y 167.648,Z 389.336,A -85,B 0,C 180,E1 -27899.758,E2 -27899.758} C_VEL
LIN {X 0,Y 166.445,Z 393.065,A -85,B 0,C 180,E1 -27900.04,E2 -27900.04} C_VEL
LIN {X 0,Y 161.647,Z 404.946,A -85,B 0,C 180,E1 -27900.781,E2 -27900.781} C_VEL
LIN {X 0,Y 155.562,Z 416.678,A -85,B 0,C 180,E1 -27901.838,E2 -27901.838} C_VEL
LIN {X 0,Y 148.795,Z 427.144,A -85,B 0,C 180,E1 -27903.128,E2 -27903.128} C_VEL
LIN {X 0,Y 141.036,Z 436.923,A -85,B 0,C 180,E1 -27904.769,E2 -27904.769} C_VEL
LIN {X 0,Y 132.692,Z 445.652,A -85,B 0,C 180,E1 -27906.783,E2 -27906.783} C_VEL
LIN {X 0,Y 124.537,Z 452.809,A -85,B 0,C 180,E1 -27909.087,E2 -27909.087} C_VEL
LIN {X 0,Y 115.062,Z 459.734,A -85,B 0,C 180,E1 -27912.264,E2 -27912.264} C_VEL
LIN {X 0,Y 105.678,Z 465.298,A -85,B 0,C 180,E1 -27916.22,E2 -27916.22} C_VEL
LIN {X 0,Y 96.197,Z 469.777,A -85,B 0,C 180,E1 -27921.407,E2 -27921.407} C_VEL
LIN {X 0,Y 87.445,Z 472.824,A -85,B 0,C 180,E1 -27927.878,E2 -27927.878} C_VEL
LIN {X 0,Y 83.024,Z 473.883,A -85,B 0,C 180,E1 -27932.182,E2 -27932.182} C_VEL
LIN {X 0,Y 77.408,Z 474.617,A -85,B 0,C 180,E1 -27939.432,E2 -27939.432} C_VEL
LIN {X 0,Y 73.066,Z 474.315,A -85,B 0,C 180,E1 -27947.689,E2 -27947.689} C_VEL
LIN {X 0,Y 71.024,Z 473.553,A -85,B 0,C 180,E1 -27953.59,E2 -27953.59} C_VEL
LIN {X 0,Y 69.651,Z 472.31,A -85,B 0,C 180,E1 -27959.712,E2 -27959.712} C_VEL
LIN {X 0,Y 68.958,Z 469.491,A -85,B 0,C 180,E1 -27969.3,E2 -27969.3} C_VEL
LIN {X 0,Y 69.725,Z 465.701,A -85,B 0,C 180,E1 -27978.379,E2 -27978.379} C_VEL
LIN {X 0,Y 71.661,Z 460.665,A -85,B 0,C 180,E1 -27987.198,E2 -27987.198} C_VEL
LIN {X 0,Y 74.69,Z 454.323,A -85,B 0,C 180,E1 -27995.408,E2 -27995.408} C_VEL
LIN {X 0,Y 78.716,Z 446.661,A -85,B 0,C 180,E1 -28002.699,E2 -28002.699} C_VEL
LIN {X 0,Y 83.28,Z 438.265,A -85,B 0,C 180,E1 -28008.457,E2 -28008.457} C_VEL
LIN {X 0,Y 88.302,Z 428.295,A -85,B 0,C 180,E1 -28013.458,E2 -28013.458} C_VEL
LIN {X 0,Y 93.362,Z 417.15,A -85,B 0,C 180,E1 -28017.463,E2 -28017.463} C_VEL
LIN {X 0,Y 97.971,Z 404.786,A -85,B 0,C 180,E1 -28020.625,E2 -28020.625} C_VEL
LIN {X 0,Y 101.608,Z 392.67,A -85,B 0,C 180,E1 -28022.816,E2 -28022.816} C_VEL
LIN {X 0,Y 104.424,Z 379.891,A -85,B 0,C 180,E1 -28024.401,E2 -28024.401} C_VEL
LIN {X 0,Y 106.439,Z 365.958,A -85,B 0,C 180,E1 -28025.429,E2 -28025.429} C_VEL
LIN {X 0,Y 109.383,Z 332.654,A -85,B 0,C 180,E1 -28027.125,E2 -28027.125} C_VEL
LIN {X 0,Y 105.185,Z 322.988,A -85,B 0,C 180,E1 -28030.958,E2 -28030.958} C_VEL
LIN {X 0,Y 100.893,Z 314.6,A -85,B 0,C 180,E1 -28035.387,E2 -28035.387} C_VEL
LIN {X 0,Y 97.195,Z 308.454,A -85,B 0,C 180,E1 -28039.87,E2 -28039.87} C_VEL
LIN {X 0,Y 94.638,Z 304.503,A -85,B 0,C 180,E1 -28043.574,E2 -28043.574} C_VEL
LIN {X 0,Y 92.019,Z 300.576,A -85,B 0,C 180,E1 -28048.187,E2 -28048.187} C_VEL
LIN {X 0,Y 89.552,Z 297.317,A -85,B 0,C 180,E1 -28053.912,E2 -28053.912} C_VEL
LIN {X 0,Y 89.039,Z 295.993,A -85,B 0,C 180,E1 -28055.654,E2 -28055.654} C_VEL
LIN {X 0,Y 86.831,Z 293.939,A -85,B 0,C 180,E1 -28068.758,E2 -28068.758} C_VEL
LIN {X 0,Y 87.841,Z 294.404,A -85,B 0,C 180,E1 -28078.585,E2 -28078.585} C_VEL
LIN {X 0,Y 89.498,Z 296.059,A -85,B 0,C 180,E1 -28084.38,E2 -28084.38} C_VEL
LIN {X 0,Y 91.376,Z 299.49,A -85,B 0,C 180,E1 -28089.276,E2 -28089.276} C_VEL
LIN {X 0,Y 92.608,Z 301.038,A -85,B 0,C 180,E1 -28091.691,E2 -28091.691} C_VEL
LIN {X 0,Y 94.921,Z 304.55,A -85,B 0,C 180,E1 -28095.627,E2 -28095.627} C_VEL
LIN {X 0,Y 98.709,Z 310.779,A -85,B 0,C 180,E1 -28100.871,E2 -28100.871} C_VEL
LIN {X 0,Y 102.684,Z 317.916,A -85,B 0,C 180,E1 -28105.367,E2 -28105.367} C_VEL
LIN {X 0,Y 106.746,Z 326.49,A -85,B 0,C 180,E1 -28109.359,E2 -28109.359} C_VEL
LIN {X 0,Y 108.503,Z 331.946,A -85,B 0,C 180,E1 -28111.09,E2 -28111.09} C_VEL
LIN {X 0,Y 109.347,Z 335.34,A -85,B 0,C 180,E1 -28111.962,E2 -28111.962} C_VEL
LIN {X 0,Y 105.753,Z 373.328,A -85,B 0,C 180,E1 -28113.899,E2 -28113.899} C_VEL
LIN {X 0,Y 103.39,Z 386.563,A -85,B 0,C 180,E1 -28115.078,E2 -28115.078} C_VEL
LIN {X 0,Y 100.384,Z 398.69,A -85,B 0,C 180,E1 -28116.789,E2 -28116.789} C_VEL
LIN {X 0,Y 96.302,Z 410.745,A -85,B 0,C 180,E1 -28119.149,E2 -28119.149} C_VEL
LIN {X 0,Y 92.804,Z 419.712,A -85,B 0,C 180,E1 -28121.588,E2 -28121.588} C_VEL
LIN {X 0,Y 88.448,Z 429.521,A -85,B 0,C 180,E1 -28125.146,E2 -28125.146} C_VEL
LIN {X 0,Y 83.799,Z 438.542,A -85,B 0,C 180,E1 -28129.451,E2 -28129.451} C_VEL
LIN {X 0,Y 80.283,Z 445.346,A -85,B 0,C 180,E1 -28133.77,E2 -28133.77} C_VEL
LIN {X 0,Y 75.762,Z 453.713,A -85,B 0,C 180,E1 -28140.846,E2 -28140.846} C_VEL
LIN {X 0,Y 72.447,Z 460.432,A -85,B 0,C 180,E1 -28148.658,E2 -28148.658} C_VEL
LIN {X 0,Y 70.231,Z 466.532,A -85,B 0,C 180,E1 -28158.446,E2 -28158.446} C_VEL
LIN {X 0,Y 69.62,Z 470.454,A -85,B 0,C 180,E1 -28167.098,E2 -28167.098} C_VEL
LIN {X 0,Y 69.677,Z 471.515,A -85,B 0,C 180,E1 -28169.991,E2 -28169.991} C_VEL
LIN {X 0,Y 69.749,Z 473.301,A -85,B 0,C 180,E1 -28175.774,E2 -28175.774} C_VEL
LIN {X 0,Y 71.489,Z 475.578,A -85,B 0,C 180,E1 -28187.144,E2 -28187.144} C_VEL
LIN {X 0,Y 75.586,Z 476.345,A -85,B 0,C 180,E1 -28197.694,E2 -28197.694} C_VEL
LIN {X 0,Y 82.055,Z 475.55,A -85,B 0,C 180,E1 -28206.828,E2 -28206.828} C_VEL
LIN {X 0,Y 90.343,Z 473.248,A -85,B 0,C 180,E1 -28214.427,E2 -28214.427} C_VEL
LIN {X 0,Y 97.502,Z 470.441,A -85,B 0,C 180,E1 -28219.177,E2 -28219.177} C_VEL
LIN {X 0,Y 105.134,Z 466.662,A -85,B 0,C 180,E1 -28223.328,E2 -28223.328} C_VEL
LIN {X 0,Y 113.345,Z 461.8,A -85,B 0,C 180,E1 -28226.821,E2 -28226.821} C_VEL
LIN {X 0,Y 121.964,Z 455.709,A -85,B 0,C 180,E1 -28229.798,E2 -28229.798} C_VEL
LIN {X 0,Y 130.907,Z 448.164,A -85,B 0,C 180,E1 -28232.343,E2 -28232.343} C_VEL
LIN {X 0,Y 140.05,Z 438.74,A -85,B 0,C 180,E1 -28234.581,E2 -28234.581} C_VEL
LIN {X 0,Y 147.94,Z 429.008,A -85,B 0,C 180,E1 -28236.121,E2 -28236.121} C_VEL
LIN {X 0,Y 155.073,Z 418.2,A -85,B 0,C 180,E1 -28237.417,E2 -28237.417} C_VEL
LIN {X 0,Y 161.218,Z 406.493,A -85,B 0,C 180,E1 -28238.442,E2 -28238.442} C_VEL
LIN {X 0,Y 166.355,Z 393.889,A -85,B 0,C 180,E1 -28239.217,E2 -28239.217} C_VEL
LIN {X 0,Y 169.852,Z 382.114,A -85,B 0,C 180,E1 -28239.743,E2 -28239.743} C_VEL
LIN {X 0,Y 169.489,Z 379.597,A -85,B 0,C 180,E1 -28241.789,E2 -28241.789} C_VEL
LIN {X 0,Y 169.158,Z 378.425,A -85,B 0,C 180,E1 -28243.396,E2 -28243.396} C_VEL
LIN {X 0,Y 168.796,Z 375.861,A -85,B 0,C 180,E1 -28247.365,E2 -28247.365} C_VEL
LIN {X 0,Y 168.95,Z 375.738,A -85,B 0,C 180,E1 -28252.822,E2 -28252.822} C_VEL
LIN {X 0,Y 169.594,Z 379.465,A -85,B 0,C 180,E1 -28257.8,E2 -28257.8} C_VEL
LIN {X 0,Y 169.937,Z 381.232,A -85,B 0,C 180,E1 -28259.425,E2 -28259.425} C_VEL
LIN {X 0,Y 166.445,Z 393.065,A -85,B 0,C 180,E1 -28260.04,E2 -28260.04} C_VEL
LIN {X 0,Y 164.235,Z 398.636,A -85,B 0,C 180,E1 -28260.126,E2 -28260.126} C_VEL
LIN {X 0,Y 157.825,Z 410.882,A -85,B 0,C 180,E1 -28259.522,E2 -28259.522} C_VEL
LIN {X 0,Y 153.712,Z 417.573,A -85,B 0,C 180,E1 -28259.432,E2 -28259.432} C_VEL
LIN {X 0,Y 151.651,Z 420.749,A -85,B 0,C 180,E1 -28259.668,E2 -28259.668} C_VEL
LIN {X 0,Y 144.084,Z 431.302,A -85,B 0,C 180,E1 -28260.999,E2 -28260.999} C_VEL
LIN {X 0,Y 135.257,Z 441.25,A -85,B 0,C 180,E1 -28262.762,E2 -28262.762} C_VEL
LIN {X 0,Y 126.915,Z 449.053,A -85,B 0,C 180,E1 -28264.678,E2 -28264.678} C_VEL
LIN {X 0,Y 117.832,Z 456.151,A -85,B 0,C 180,E1 -28267.155,E2 -28267.155} C_VEL
LIN {X 0,Y 110.45,Z 460.987,A -85,B 0,C 180,E1 -28269.542,E2 -28269.542} C_VEL
LIN {X 0,Y 101.072,Z 466.119,A -85,B 0,C 180,E1 -28273.252,E2 -28273.252} C_VEL
LIN {X 0,Y 92.275,Z 469.952,A -85,B 0,C 180,E1 -28277.719,E2 -28277.719} C_VEL
LIN {X 0,Y 84.074,Z 472.65,A -85,B 0,C 180,E1 -28283.163,E2 -28283.163} C_VEL
LIN {X 0,Y 79.125,Z 473.813,A -85,B 0,C 180,E1 -28287.369,E2 -28287.369} C_VEL
LIN {X 0,Y 71.765,Z 474.725,A -85,B 0,C 180,E1 -28295.957,E2 -28295.957} C_VEL
LIN {X 0,Y 67.514,Z 474.529,A -85,B 0,C 180,E1 -28303.238,E2 -28303.238} C_VEL
LIN {X 0,Y 64.96,Z 473.837,A -85,B 0,C 180,E1 -28309.537,E2 -28309.537} C_VEL
LIN {X 0,Y 63.111,Z 472.718,A -85,B 0,C 180,E1 -28316.178,E2 -28316.178} C_VEL
LIN {X 0,Y 61.963,Z 470.545,A -85,B 0,C 180,E1 -28325.08,E2 -28325.08} C_VEL
LIN {X 0,Y 62.398,Z 466.434,A -85,B 0,C 180,E1 -28336.992,E2 -28336.992} C_VEL
LIN {X 0,Y 64.327,Z 461.48,A -85,B 0,C 180,E1 -28347.016,E2 -28347.016} C_VEL
LIN {X 0,Y 67.346,Z 455.408,A -85,B 0,C 180,E1 -28355.999,E2 -28355.999} C_VEL
LIN {X 0,Y 71.738,Z 447.725,A -85,B 0,C 180,E1 -28364.189,E2 -28364.189} C_VEL
LIN {X 0,Y 76.449,Z 439.84,A -85,B 0,C 180,E1 -28370.174,E2 -28370.174} C_VEL
LIN {X 0,Y 81.678,Z 430.246,A -85,B 0,C 180,E1 -28375.49,E2 -28375.49} C_VEL
LIN {X 0,Y 86.983,Z 419.493,A -85,B 0,C 180,E1 -28379.67,E2 -28379.67} C_VEL
LIN {X 0,Y 91.921,Z 407.58,A -85,B 0,C 180,E1 -28383,E2 -28383} C_VEL
LIN {X 0,Y 95.975,Z 395.284,A -85,B 0,C 180,E1 -28385.39,E2 -28385.39} C_VEL
LIN {X 0,Y 99.25,Z 382.06,A -85,B 0,C 180,E1 -28387.155,E2 -28387.155} C_VEL
LIN {X 0,Y 101.32,Z 369.967,A -85,B 0,C 180,E1 -28388.158,E2 -28388.158} C_VEL
LIN {X 0,Y 104.674,Z 335.069,A -85,B 0,C 180,E1 -28389.929,E2 -28389.929} C_VEL
LIN {X 0,Y 100.585,Z 325.499,A -85,B 0,C 180,E1 -28394.21,E2 -28394.21} C_VEL
LIN {X 0,Y 96.882,Z 318.138,A -85,B 0,C 180,E1 -28398.688,E2 -28398.688} C_VEL
LIN {X 0,Y 94.253,Z 313.682,A -85,B 0,C 180,E1 -28402.395,E2 -28402.395} C_VEL
LIN {X 0,Y 92.438,Z 310.629,A -85,B 0,C 180,E1 -28405.403,E2 -28405.403} C_VEL
LIN {X 0,Y 90.263,Z 307.076,A -85,B 0,C 180,E1 -28409.698,E2 -28409.698} C_VEL
LIN {X 0,Y 88.057,Z 303.794,A -85,B 0,C 180,E1 -28415.507,E2 -28415.507} C_VEL
LIN {X 0,Y 87.656,Z 302.855,A -85,B 0,C 180,E1 -28417.012,E2 -28417.012} C_VEL
LIN {X 0,Y 85.927,Z 300.955,A -85,B 0,C 180,E1 -28428.993,E2 -28428.993} C_VEL
LIN {X 0,Y 86.913,Z 301.499,A -85,B 0,C 180,E1 -28438.57,E2 -28438.57} C_VEL
LIN {X 0,Y 88.134,Z 302.949,A -85,B 0,C 180,E1 -28443.232,E2 -28443.232} C_VEL
LIN {X 0,Y 90.238,Z 306.666,A -85,B 0,C 180,E1 -28448.978,E2 -28448.978} C_VEL
LIN {X 0,Y 91.289,Z 308.547,A -85,B 0,C 180,E1 -28451.242,E2 -28451.242} C_VEL
LIN {X 0,Y 93.317,Z 311.826,A -85,B 0,C 180,E1 -28454.881,E2 -28454.881} C_VEL
LIN {X 0,Y 96.529,Z 317.323,A -85,B 0,C 180,E1 -28459.642,E2 -28459.642} C_VEL
LIN {X 0,Y 100.644,Z 325.634,A -85,B 0,C 180,E1 -28464.683,E2 -28464.683} C_VEL
LIN {X 0,Y 103.558,Z 332.689,A -85,B 0,C 180,E1 -28467.823,E2 -28467.823} C_VEL
LIN {X 0,Y 104.648,Z 337.619,A -85,B 0,C 180,E1 -28469.173,E2 -28469.173} C_VEL
LIN {X 0,Y 101.092,Z 373.069,A -85,B 0,C 180,E1 -28470.941,E2 -28470.941} C_VEL
LIN {X 0,Y 98.725,Z 385.835,A -85,B 0,C 180,E1 -28472.039,E2 -28472.039} C_VEL
LIN {X 0,Y 95.594,Z 398.006,A -85,B 0,C 180,E1 -28473.717,E2 -28473.717} C_VEL
LIN {X 0,Y 91.313,Z 410.24,A -85,B 0,C 180,E1 -28476.074,E2 -28476.074} C_VEL
LIN {X 0,Y 87.593,Z 419.272,A -85,B 0,C 180,E1 -28478.519,E2 -28478.519} C_VEL
LIN {X 0,Y 82.936,Z 429.143,A -85,B 0,C 180,E1 -28482.134,E2 -28482.134} C_VEL
LIN {X 0,Y 77.325,Z 439.449,A -85,B 0,C 180,E1 -28487.332,E2 -28487.332} C_VEL
LIN {X 0,Y 72.837,Z 447.318,A -85,B 0,C 180,E1 -28492.9,E2 -28492.9} C_VEL
LIN {X 0,Y 68.183,Z 455.313,A -85,B 0,C 180,E1 -28500.675,E2 -28500.675} C_VEL
LIN {X 0,Y 65.373,Z 460.715,A -85,B 0,C 180,E1 -28507.887,E2 -28507.887} C_VEL
LIN {X 0,Y 63.286,Z 465.967,A -85,B 0,C 180,E1 -28517.157,E2 -28517.157} C_VEL
LIN {X 0,Y 62.527,Z 470.003,A -85,B 0,C 180,E1 -28526.768,E2 -28526.768} C_VEL
LIN {X 0,Y 62.605,Z 471.082,A -85,B 0,C 180,E1 -28529.99,E2 -28529.99} C_VEL
LIN {X 0,Y 62.697,Z 472.934,A -85,B 0,C 180,E1 -28536.426,E2 -28536.426} C_VEL
LIN {X 0,Y 63.357,Z 474.35,A -85,B 0,C 180,E1 -28542.808,E2 -28542.808} C_VEL
LIN {X 0,Y 66.715,Z 475.968,A -85,B 0,C 180,E1 -28554.911,E2 -28554.911} C_VEL
LIN {X 0,Y 72.633,Z 476.105,A -85,B 0,C 180,E1 -28565.479,E2 -28565.479} C_VEL
LIN {X 0,Y 80.757,Z 474.679,A -85,B 0,C 180,E1 -28574.113,E2 -28574.113} C_VEL
LIN {X 0,Y 90.437,Z 471.719,A -85,B 0,C 180,E1 -28580.985,E2 -28580.985} C_VEL
LIN {X 0,Y 98.052,Z 468.506,A -85,B 0,C 180,E1 -28585.142,E2 -28585.142} C_VEL
LIN {X 0,Y 106.726,Z 464.02,A -85,B 0,C 180,E1 -28588.865,E2 -28588.865} C_VEL
LIN {X 0,Y 115.579,Z 458.497,A -85,B 0,C 180,E1 -28591.835,E2 -28591.835} C_VEL
LIN {X 0,Y 124.739,Z 451.629,A -85,B 0,C 180,E1 -28594.338,E2 -28594.338} C_VEL
LIN {X 0,Y 132.462,Z 444.671,A -85,B 0,C 180,E1 -28596.225,E2 -28596.225} C_VEL
LIN {X 0,Y 140.402,Z 436.284,A -85,B 0,C 180,E1 -28597.813,E2 -28597.813} C_VEL
LIN {X 0,Y 148.467,Z 425.981,A -85,B 0,C 180,E1 -28599.2,E2 -28599.2} C_VEL
LIN {X 0,Y 155.774,Z 414.459,A -85,B 0,C 180,E1 -28600.345,E2 -28600.345} C_VEL
LIN {X 0,Y 161.729,Z 402.488,A -85,B 0,C 180,E1 -28601.191,E2 -28601.191} C_VEL
LIN {X 0,Y 166.341,Z 390.341,A -85,B 0,C 180,E1 -28601.774,E2 -28601.774} C_VEL
LIN {X 0,Y 167.5,Z 386.566,A -85,B 0,C 180,E1 -28601.953,E2 -28601.953} C_VEL
LIN {X 0,Y 167.276,Z 385.244,A -85,B 0,C 180,E1 -28603.595,E2 -28603.595} C_VEL
LIN {X 0,Y 167.086,Z 382.673,A -85,B 0,C 180,E1 -28607.85,E2 -28607.85} C_VEL
LIN {X 0,Y 167.211,Z 382.772,A -85,B 0,C 180,E1 -28612.747,E2 -28612.747} C_VEL
LIN {X 0,Y 167.511,Z 385.996,A -85,B 0,C 180,E1 -28617.158,E2 -28617.158} C_VEL
LIN {X 0,Y 167.526,Z 386.141,A -85,B 0,C 180,E1 -28617.301,E2 -28617.301} C_VEL
LIN {X 0,Y 163.163,Z 398.672,A -85,B 0,C 180,E1 -28617.909,E2 -28617.909} C_VEL
LIN {X 0,Y 158.162,Z 409.525,A -85,B 0,C 180,E1 -28618.634,E2 -28618.634} C_VEL
LIN {X 0,Y 151.651,Z 420.749,A -85,B 0,C 180,E1 -28619.668,E2 -28619.668} C_VEL
LIN {X 0,Y 148.31,Z 425.549,A -85,B 0,C 180,E1 -28619.993,E2 -28619.993} C_VEL
LIN {X 0,Y 141.943,Z 433.159,A -85,B 0,C 180,E1 -28619.892,E2 -28619.892} C_VEL
LIN {X 0,Y 135.015,Z 440.236,A -85,B 0,C 180,E1 -28619.852,E2 -28619.852} C_VEL
LIN {X 0,Y 130.799,Z 444.2,A -85,B 0,C 180,E1 -28620.339,E2 -28620.339} C_VEL
LIN {X 0,Y 121.325,Z 452.213,A -85,B 0,C 180,E1 -28622.373,E2 -28622.373} C_VEL
LIN {X 0,Y 111.108,Z 459.283,A -85,B 0,C 180,E1 -28625.039,E2 -28625.039} C_VEL
LIN {X 0,Y 102.34,Z 464.239,A -85,B 0,C 180,E1 -28627.879,E2 -28627.879} C_VEL
LIN {X 0,Y 93.24,Z 468.421,A -85,B 0,C 180,E1 -28631.548,E2 -28631.548} C_VEL
LIN {X 0,Y 87.132,Z 470.686,A -85,B 0,C 180,E1 -28634.585,E2 -28634.585} C_VEL
LIN {X 0,Y 76.566,Z 473.568,A -85,B 0,C 180,E1 -28641.518,E2 -28641.518} C_VEL
LIN {X 0,Y 70.823,Z 474.508,A -85,B 0,C 180,E1 -28646.755,E2 -28646.755} C_VEL
LIN {X 0,Y 66.324,Z 474.837,A -85,B 0,C 180,E1 -28652.055,E2 -28652.055} C_VEL
LIN {X 0,Y 62.421,Z 474.731,A -85,B 0,C 180,E1 -28658.006,E2 -28658.006} C_VEL
LIN {X 0,Y 58.845,Z 473.984,A -85,B 0,C 180,E1 -28665.734,E2 -28665.734} C_VEL
LIN {X 0,Y 55.367,Z 471.579,A -85,B 0,C 180,E1 -28679.5,E2 -28679.5} C_VEL
LIN {X 0,Y 54.824,Z 468.404,A -85,B 0,C 180,E1 -28691.32,E2 -28691.32} C_VEL
LIN {X 0,Y 56.121,Z 464.087,A -85,B 0,C 180,E1 -28702.817,E2 -28702.817} C_VEL
LIN {X 0,Y 58.949,Z 458.54,A -85,B 0,C 180,E1 -28713.428,E2 -28713.428} C_VEL
LIN {X 0,Y 63.075,Z 451.615,A -85,B 0,C 180,E1 -28722.886,E2 -28722.886} C_VEL
LIN {X 0,Y 67.968,Z 443.991,A -85,B 0,C 180,E1 -28730.198,E2 -28730.198} C_VEL
LIN {X 0,Y 72.888,Z 435.979,A -85,B 0,C 180,E1 -28735.725,E2 -28735.725} C_VEL
LIN {X 0,Y 78.23,Z 426.598,A -85,B 0,C 180,E1 -28740.363,E2 -28740.363} C_VEL
LIN {X 0,Y 83.322,Z 416.336,A -85,B 0,C 180,E1 -28743.982,E2 -28743.982} C_VEL
LIN {X 0,Y 88.262,Z 404.344,A -85,B 0,C 180,E1 -28747.005,E2 -28747.005} C_VEL
LIN {X 0,Y 92.379,Z 391.762,A -85,B 0,C 180,E1 -28749.188,E2 -28749.188} C_VEL
LIN {X 0,Y 95.465,Z 378.555,A -85,B 0,C 180,E1 -28750.711,E2 -28750.711} C_VEL
LIN {X 0,Y 97.441,Z 365.513,A -85,B 0,C 180,E1 -28751.609,E2 -28751.609} C_VEL
LIN {X 0,Y 100.187,Z 337.682,A -85,B 0,C 180,E1 -28752.969,E2 -28752.969} C_VEL
LIN {X 0,Y 96.983,Z 329.829,A -85,B 0,C 180,E1 -28756.841,E2 -28756.841} C_VEL
LIN {X 0,Y 93.927,Z 323.213,A -85,B 0,C 180,E1 -28761.124,E2 -28761.124} C_VEL
LIN {X 0,Y 90.7,Z 317.247,A -85,B 0,C 180,E1 -28766.618,E2 -28766.618} C_VEL
LIN {X 0,Y 88.569,Z 313.606,A -85,B 0,C 180,E1 -28771.267,E2 -28771.267} C_VEL
LIN {X 0,Y 86.536,Z 310.013,A -85,B 0,C 180,E1 -28777.565,E2 -28777.565} C_VEL
LIN {X 0,Y 85.019,Z 308.024,A -85,B 0,C 180,E1 -28788.816,E2 -28788.816} C_VEL
LIN {X 0,Y 85.808,Z 308.438,A -85,B 0,C 180,E1 -28797.671,E2 -28797.671} C_VEL
LIN {X 0,Y 86.803,Z 309.781,A -85,B 0,C 180,E1 -28802.012,E2 -28802.012} C_VEL
LIN {X 0,Y 89.088,Z 314.094,A -85,B 0,C 180,E1 -28808.712,E2 -28808.712} C_VEL
LIN {X 0,Y 91.326,Z 318.261,A -85,B 0,C 180,E1 -28813.365,E2 -28813.365} C_VEL
LIN {X 0,Y 94.094,Z 323.465,A -85,B 0,C 180,E1 -28817.942,E2 -28817.942} C_VEL
LIN {X 0,Y 97.707,Z 331.499,A -85,B 0,C 180,E1 -28822.901,E2 -28822.901} C_VEL
LIN {X 0,Y 99.786,Z 336.962,A -85,B 0,C 180,E1 -28825.438,E2 -28825.438} C_VEL
LIN {X 0,Y 100.238,Z 338.872,A -85,B 0,C 180,E1 -28826.048,E2 -28826.048} C_VEL
LIN {X 0,Y 96.617,Z 373.309,A -85,B 0,C 180,E1 -28827.758,E2 -28827.758} C_VEL
LIN {X 0,Y 94.064,Z 386.349,A -85,B 0,C 180,E1 -28828.875,E2 -28828.875} C_VEL
LIN {X 0,Y 90.778,Z 398.363,A -85,B 0,C 180,E1 -28830.525,E2 -28830.525} C_VEL
LIN {X 0,Y 86.619,Z 409.658,A -85,B 0,C 180,E1 -28832.657,E2 -28832.657} C_VEL
LIN {X 0,Y 82.668,Z 418.75,A -85,B 0,C 180,E1 -28835.076,E2 -28835.076} C_VEL
LIN {X 0,Y 77.701,Z 428.71,A -85,B 0,C 180,E1 -28838.715,E2 -28838.715} C_VEL
LIN {X 0,Y 73.103,Z 436.674,A -85,B 0,C 180,E1 -28842.572,E2 -28842.572} C_VEL
LIN {X 0,Y 68.248,Z 444.715,A -85,B 0,C 180,E1 -28847.971,E2 -28847.971} C_VEL
LIN {X 0,Y 62.856,Z 453.164,A -85,B 0,C 180,E1 -28855.998,E2 -28855.998} C_VEL
LIN {X 0,Y 58.811,Z 459.944,A -85,B 0,C 180,E1 -28865.264,E2 -28865.264} C_VEL
LIN {X 0,Y 56.363,Z 465.331,A -85,B 0,C 180,E1 -28875.548,E2 -28875.548} C_VEL
LIN {X 0,Y 55.452,Z 469.49,A -85,B 0,C 180,E1 -28886.355,E2 -28886.355} C_VEL
LIN {X 0,Y 55.514,Z 470.626,A -85,B 0,C 180,E1 -28889.989,E2 -28889.989} C_VEL
LIN {X 0,Y 55.646,Z 472.534,A -85,B 0,C 180,E1 -28897.244,E2 -28897.244} C_VEL
LIN {X 0,Y 56.456,Z 474.031,A -85,B 0,C 180,E1 -28904.405,E2 -28904.405} C_VEL
LIN {X 0,Y 58.053,Z 475.112,A -85,B 0,C 180,E1 -28911.284,E2 -28911.284} C_VEL
LIN {X 0,Y 63.308,Z 476.094,A -85,B 0,C 180,E1 -28923.703,E2 -28923.703} C_VEL
LIN {X 0,Y 71.196,Z 475.607,A -85,B 0,C 180,E1 -28933.696,E2 -28933.696} C_VEL
LIN {X 0,Y 80.824,Z 473.54,A -85,B 0,C 180,E1 -28941.485,E2 -28941.485} C_VEL
LIN {X 0,Y 91.638,Z 469.905,A -85,B 0,C 180,E1 -28947.512,E2 -28947.512} C_VEL
LIN {X 0,Y 100.285,Z 466.011,A -85,B 0,C 180,E1 -28951.149,E2 -28951.149} C_VEL
LIN {X 0,Y 109.318,Z 461.028,A -85,B 0,C 180,E1 -28954.15,E2 -28954.15} C_VEL
LIN {X 0,Y 118.683,Z 454.805,A -85,B 0,C 180,E1 -28956.6,E2 -28956.6} C_VEL
LIN {X 0,Y 128.176,Z 447.08,A -85,B 0,C 180,E1 -28958.753,E2 -28958.753} C_VEL
LIN {X 0,Y 136.255,Z 439.231,A -85,B 0,C 180,E1 -28960.262,E2 -28960.262} C_VEL
LIN {X 0,Y 144.49,Z 429.655,A -85,B 0,C 180,E1 -28961.513,E2 -28961.513} C_VEL
LIN {X 0,Y 151.914,Z 419.093,A -85,B 0,C 180,E1 -28962.571,E2 -28962.571} C_VEL
LIN {X 0,Y 158.435,Z 407.448,A -85,B 0,C 180,E1 -28963.421,E2 -28963.421} C_VEL
LIN {X 0,Y 163.734,Z 395.224,A -85,B 0,C 180,E1 -28964.038,E2 -28964.038} C_VEL
LIN {X 0,Y 164.751,Z 392.478,A -85,B 0,C 180,E1 -28964.133,E2 -28964.133} C_VEL
LIN {X 0,Y 164.948,Z 391.552,A -85,B 0,C 180,E1 -28964.547,E2 -28964.547} C_VEL
LIN {X 0,Y 164.969,Z 389.414,A -85,B 0,C 180,E1 -28968.455,E2 -28968.455} C_VEL
LIN {X 0,Y 165.07,Z 389.666,A -85,B 0,C 180,E1 -28972.652,E2 -28972.652} C_VEL
LIN {X 0,Y 164.938,Z 391.642,A -85,B 0,C 180,E1 -28975.102,E2 -28975.102} C_VEL
LIN {X 0,Y 160.334,Z 403.181,A -85,B 0,C 180,E1 -28975.662,E2 -28975.662} C_VEL
LIN {X 0,Y 154.915,Z 413.727,A -85,B 0,C 180,E1 -28976.364,E2 -28976.364} C_VEL
LIN {X 0,Y 147.726,Z 424.91,A -85,B 0,C 180,E1 -28977.416,E2 -28977.416} C_VEL
LIN {X 0,Y 139.705,Z 435.034,A -85,B 0,C 180,E1 -28978.7,E2 -28978.7} C_VEL
LIN {X 0,Y 130.799,Z 444.2,A -85,B 0,C 180,E1 -28980.339,E2 -28980.339} C_VEL
LIN {X 0,Y 126.409,Z 448.01,A -85,B 0,C 180,E1 -28980.904,E2 -28980.904} C_VEL
LIN {X 0,Y 118.413,Z 453.875,A -85,B 0,C 180,E1 -28981.176,E2 -28981.176} C_VEL
LIN {X 0,Y 110.055,Z 459.066,A -85,B 0,C 180,E1 -28981.602,E2 -28981.602} C_VEL
LIN {X 0,Y 105.135,Z 461.79,A -85,B 0,C 180,E1 -28982.516,E2 -28982.516} C_VEL
LIN {X 0,Y 95.319,Z 466.626,A -85,B 0,C 180,E1 -28985.585,E2 -28985.585} C_VEL
LIN {X 0,Y 85.505,Z 470.388,A -85,B 0,C 180,E1 -28989.532,E2 -28989.532} C_VEL
LIN {X 0,Y 79.241,Z 472.222,A -85,B 0,C 180,E1 -28992.719,E2 -28992.719} C_VEL
LIN {X 0,Y 72.655,Z 473.713,A -85,B 0,C 180,E1 -28996.847,E2 -28996.847} C_VEL
LIN {X 0,Y 67.654,Z 474.505,A -85,B 0,C 180,E1 -29000.81,E2 -29000.81} C_VEL
LIN {X 0,Y 61.447,Z 474.942,A -85,B 0,C 180,E1 -29007.196,E2 -29007.196} C_VEL
LIN {X 0,Y 54.082,Z 474.402,A -85,B 0,C 180,E1 -29018.785,E2 -29018.785} C_VEL
LIN {X 0,Y 51.025,Z 473.423,A -85,B 0,C 180,E1 -29026.491,E2 -29026.491} C_VEL
LIN {X 0,Y 48.044,Z 470.698,A -85,B 0,C 180,E1 -29041.294,E2 -29041.294} C_VEL
LIN {X 0,Y 47.791,Z 467.716,A -85,B 0,C 180,E1 -29052.91,E2 -29052.91} C_VEL
LIN {X 0,Y 49.344,Z 463.493,A -85,B 0,C 180,E1 -29065.143,E2 -29065.143} C_VEL
LIN {X 0,Y 52.86,Z 457.386,A -85,B 0,C 180,E1 -29077.652,E2 -29077.652} C_VEL
LIN {X 0,Y 57.767,Z 450.162,A -85,B 0,C 180,E1 -29087.718,E2 -29087.718} C_VEL
LIN {X 0,Y 63.208,Z 442.441,A -85,B 0,C 180,E1 -29094.953,E2 -29094.953} C_VEL
LIN {X 0,Y 69.475,Z 432.724,A -85,B 0,C 180,E1 -29101.238,E2 -29101.238} C_VEL
LIN {X 0,Y 75.339,Z 422.604,A -85,B 0,C 180,E1 -29105.674,E2 -29105.674} C_VEL
LIN {X 0,Y 80.533,Z 412.073,A -85,B 0,C 180,E1 -29108.895,E2 -29108.895} C_VEL
LIN {X 0,Y 85.124,Z 400.722,A -85,B 0,C 180,E1 -29111.347,E2 -29111.347} C_VEL
LIN {X 0,Y 88.96,Z 388.493,A -85,B 0,C 180,E1 -29113.21,E2 -29113.21} C_VEL
LIN {X 0,Y 91.98,Z 375.225,A -85,B 0,C 180,E1 -29114.481,E2 -29114.481} C_VEL
LIN {X 0,Y 94.129,Z 358.251,A -85,B 0,C 180,E1 -29115.434,E2 -29115.434} C_VEL
LIN {X 0,Y 95.953,Z 340.238,A -85,B 0,C 180,E1 -29116.315,E2 -29116.315} C_VEL
LIN {X 0,Y 93.234,Z 333.121,A -85,B 0,C 180,E1 -29120.25,E2 -29120.25} C_VEL
LIN {X 0,Y 90.403,Z 326.784,A -85,B 0,C 180,E1 -29125.07,E2 -29125.07} C_VEL
LIN {X 0,Y 88.279,Z 322.717,A -85,B 0,C 180,E1 -29129.435,E2 -29129.435} C_VEL
LIN {X 0,Y 86.886,Z 320,A -85,B 0,C 180,E1 -29133.048,E2 -29133.048} C_VEL
LIN {X 0,Y 85.075,Z 316.484,A -85,B 0,C 180,E1 -29139.782,E2 -29139.782} C_VEL
LIN {X 0,Y 84.13,Z 314.993,A -85,B 0,C 180,E1 -29150.401,E2 -29150.401} C_VEL
LIN {X 0,Y 84.96,Z 315.651,A -85,B 0,C 180,E1 -29158.093,E2 -29158.093} C_VEL
LIN {X 0,Y 85.523,Z 316.579,A -85,B 0,C 180,E1 -29160.777,E2 -29160.777} C_VEL
LIN {X 0,Y 87.386,Z 320.549,A -85,B 0,C 180,E1 -29167.038,E2 -29167.038} C_VEL
LIN {X 0,Y 89.316,Z 324.545,A -85,B 0,C 180,E1 -29171.62,E2 -29171.62} C_VEL
LIN {X 0,Y 91.549,Z 329.089,A -85,B 0,C 180,E1 -29175.8,E2 -29175.8} C_VEL
LIN {X 0,Y 94.622,Z 336.679,A -85,B 0,C 180,E1 -29180.659,E2 -29180.659} C_VEL
LIN {X 0,Y 96.077,Z 340.864,A -85,B 0,C 180,E1 -29182.717,E2 -29182.717} C_VEL
LIN {X 0,Y 92.514,Z 373.08,A -85,B 0,C 180,E1 -29184.257,E2 -29184.257} C_VEL
LIN {X 0,Y 89.95,Z 385.649,A -85,B 0,C 180,E1 -29185.246,E2 -29185.246} C_VEL
LIN {X 0,Y 86.267,Z 398.621,A -85,B 0,C 180,E1 -29186.979,E2 -29186.979} C_VEL
LIN {X 0,Y 81.531,Z 410.595,A -85,B 0,C 180,E1 -29189.202,E2 -29189.202} C_VEL
LIN {X 0,Y 76.041,Z 422.153,A -85,B 0,C 180,E1 -29192.489,E2 -29192.489} C_VEL
LIN {X 0,Y 70.254,Z 432.575,A -85,B 0,C 180,E1 -29196.828,E2 -29196.828} C_VEL
LIN {X 0,Y 65.372,Z 440.159,A -85,B 0,C 180,E1 -29201.174,E2 -29201.174} C_VEL
LIN {X 0,Y 59.969,Z 448.141,A -85,B 0,C 180,E1 -29207.621,E2 -29207.621} C_VEL
LIN {X 0,Y 54.512,Z 455.881,A -85,B 0,C 180,E1 -29216.761,E2 -29216.761} C_VEL
LIN {X 0,Y 50.3,Z 463.005,A -85,B 0,C 180,E1 -29229.542,E2 -29229.542} C_VEL
LIN {X 0,Y 48.563,Z 467.691,A -85,B 0,C 180,E1 -29241.666,E2 -29241.666} C_VEL
LIN {X 0,Y 48.44,Z 470.17,A -85,B 0,C 180,E1 -29249.987,E2 -29249.987} C_VEL
LIN {X 0,Y 48.613,Z 472.134,A -85,B 0,C 180,E1 -29258.299,E2 -29258.299} C_VEL
LIN {X 0,Y 51.483,Z 474.851,A -85,B 0,C 180,E1 -29274.162,E2 -29274.162} C_VEL
LIN {X 0,Y 54.153,Z 475.608,A -85,B 0,C 180,E1 -29281.259,E2 -29281.259} C_VEL
LIN {X 0,Y 61.627,Z 475.964,A -85,B 0,C 180,E1 -29293.162,E2 -29293.162} C_VEL
LIN {X 0,Y 71.23,Z 474.847,A -85,B 0,C 180,E1 -29302.108,E2 -29302.108} C_VEL
LIN {X 0,Y 82.238,Z 472.125,A -85,B 0,C 180,E1 -29308.699,E2 -29308.699} C_VEL
LIN {X 0,Y 90.986,Z 469.036,A -85,B 0,C 180,E1 -29312.643,E2 -29312.643} C_VEL
LIN {X 0,Y 100.138,Z 464.936,A -85,B 0,C 180,E1 -29315.82,E2 -29315.82} C_VEL
LIN {X 0,Y 109.627,Z 459.7,A -85,B 0,C 180,E1 -29318.351,E2 -29318.351} C_VEL
LIN {X 0,Y 119.308,Z 453.167,A -85,B 0,C 180,E1 -29320.459,E2 -29320.459} C_VEL
LIN {X 0,Y 129.094,Z 445.107,A -85,B 0,C 180,E1 -29322.292,E2 -29322.292} C_VEL
LIN {X 0,Y 137.393,Z 436.873,A -85,B 0,C 180,E1 -29323.54,E2 -29323.54} C_VEL
LIN {X 0,Y 145.768,Z 426.788,A -85,B 0,C 180,E1 -29324.62,E2 -29324.62} C_VEL
LIN {X 0,Y 153.273,Z 415.569,A -85,B 0,C 180,E1 -29325.504,E2 -29325.504} C_VEL
LIN {X 0,Y 159.246,Z 404.39,A -85,B 0,C 180,E1 -29326.131,E2 -29326.131} C_VEL
LIN {X 0,Y 161.935,Z 398.312,A -85,B 0,C 180,E1 -29326.406,E2 -29326.406} C_VEL
LIN {X 0,Y 162.383,Z 396.986,A -85,B 0,C 180,E1 -29326.857,E2 -29326.857} C_VEL
LIN {X 0,Y 162.446,Z 396.583,A -85,B 0,C 180,E1 -29327.498,E2 -29327.498} C_VEL
LIN {X 0,Y 162.51,Z 395.997,A -85,B 0,C 180,E1 -29330.029,E2 -29330.029} C_VEL
LIN {X 0,Y 162.541,Z 396.48,A -85,B 0,C 180,E1 -29332.537,E2 -29332.537} C_VEL
LIN {X 0,Y 162.352,Z 397.085,A -85,B 0,C 180,E1 -29332.841,E2 -29332.841} C_VEL
LIN {X 0,Y 157.337,Z 408.09,A -85,B 0,C 180,E1 -29333.372,E2 -29333.372} C_VEL
LIN {X 0,Y 151.004,Z 419.013,A -85,B 0,C 180,E1 -29334.126,E2 -29334.126} C_VEL
LIN {X 0,Y 142.798,Z 430.32,A -85,B 0,C 180,E1 -29335.199,E2 -29335.199} C_VEL
LIN {X 0,Y 135.566,Z 438.497,A -85,B 0,C 180,E1 -29336.255,E2 -29336.255} C_VEL
LIN {X 0,Y 126.59,Z 446.985,A -85,B 0,C 180,E1 -29337.746,E2 -29337.746} C_VEL
LIN {X 0,Y 117.068,Z 454.385,A -85,B 0,C 180,E1 -29339.618,E2 -29339.618} C_VEL
LIN {X 0,Y 108.959,Z 459.632,A -85,B 0,C 180,E1 -29341.489,E2 -29341.489} C_VEL
LIN {X 0,Y 105.135,Z 461.79,A -85,B 0,C 180,E1 -29342.516,E2 -29342.516} C_VEL
LIN {X 0,Y 100.11,Z 464.335,A -85,B 0,C 180,E1 -29343.569,E2 -29343.569} C_VEL
LIN {X 0,Y 87.364,Z 469.303,A -85,B 0,C 180,E1 -29344.989,E2 -29344.989} C_VEL
LIN {X 0,Y 80.062,Z 471.473,A -85,B 0,C 180,E1 -29346.401,E2 -29346.401} C_VEL
LIN {X 0,Y 76.649,Z 472.297,A -85,B 0,C 180,E1 -29347.689,E2 -29347.689} C_VEL
LIN {X 0,Y 65.287,Z 474.45,A -85,B 0,C 180,E1 -29354.384,E2 -29354.384} C_VEL
LIN {X 0,Y 57.007,Z 475.05,A -85,B 0,C 180,E1 -29361.676,E2 -29361.676} C_VEL
LIN {X 0,Y 49.561,Z 474.627,A -85,B 0,C 180,E1 -29371.723,E2 -29371.723} C_VEL
LIN {X 0,Y 45.711,Z 473.778,A -85,B 0,C 180,E1 -29379.78,E2 -29379.78} C_VEL
LIN {X 0,Y 42.808,Z 472.432,A -85,B 0,C 180,E1 -29388.971,E2 -29388.971} C_VEL
LIN {X 0,Y 40.722,Z 469.545,A -85,B 0,C 180,E1 -29404.457,E2 -29404.457} C_VEL
LIN {X 0,Y 41.332,Z 465.541,A -85,B 0,C 180,E1 -29420.225,E2 -29420.225} C_VEL
LIN {X 0,Y 44.232,Z 460.349,A -85,B 0,C 180,E1 -29434.571,E2 -29434.571} C_VEL
LIN {X 0,Y 48.948,Z 453.839,A -85,B 0,C 180,E1 -29446.701,E2 -29446.701} C_VEL
LIN {X 0,Y 54.552,Z 446.512,A -85,B 0,C 180,E1 -29455.673,E2 -29455.673} C_VEL
LIN {X 0,Y 60.14,Z 439.103,A -85,B 0,C 180,E1 -29461.739,E2 -29461.739} C_VEL
LIN {X 0,Y 66.761,Z 429.229,A -85,B 0,C 180,E1 -29467.262,E2 -29467.262} C_VEL
LIN {X 0,Y 73.187,Z 418.216,A -85,B 0,C 180,E1 -29471.326,E2 -29471.326} C_VEL
LIN {X 0,Y 78.276,Z 407.64,A -85,B 0,C 180,E1 -29474.038,E2 -29474.038} C_VEL
LIN {X 0,Y 82.858,Z 395.736,A -85,B 0,C 180,E1 -29476.145,E2 -29476.145} C_VEL
LIN {X 0,Y 86.649,Z 382.493,A -85,B 0,C 180,E1 -29477.743,E2 -29477.743} C_VEL
LIN {X 0,Y 89.074,Z 370.028,A -85,B 0,C 180,E1 -29478.648,E2 -29478.648} C_VEL
LIN {X 0,Y 92.004,Z 344.082,A -85,B 0,C 180,E1 -29479.817,E2 -29479.817} C_VEL
LIN {X 0,Y 91.931,Z 342.559,A -85,B 0,C 180,E1 -29480.159,E2 -29480.159} C_VEL
LIN {X 0,Y 89.551,Z 335.904,A -85,B 0,C 180,E1 -29484.442,E2 -29484.442} C_VEL
LIN {X 0,Y 87.411,Z 331.019,A -85,B 0,C 180,E1 -29488.952,E2 -29488.952} C_VEL
LIN {X 0,Y 85.479,Z 326.714,A -85,B 0,C 180,E1 -29494.27,E2 -29494.27} C_VEL
LIN {X 0,Y 84.005,Z 323.445,A -85,B 0,C 180,E1 -29500.47,E2 -29500.47} C_VEL
LIN {X 0,Y 83.22,Z 322.044,A -85,B 0,C 180,E1 -29510.295,E2 -29510.295} C_VEL
LIN {X 0,Y 83.946,Z 322.668,A -85,B 0,C 180,E1 -29517.62,E2 -29517.62} C_VEL
LIN {X 0,Y 84.346,Z 323.591,A -85,B 0,C 180,E1 -29519.854,E2 -29519.854} C_VEL
LIN {X 0,Y 85.796,Z 327.067,A -85,B 0,C 180,E1 -29525.451,E2 -29525.451} C_VEL
LIN {X 0,Y 87.533,Z 331.121,A -85,B 0,C 180,E1 -29530.12,E2 -29530.12} C_VEL
LIN {X 0,Y 89.441,Z 335.561,A -85,B 0,C 180,E1 -29534.159,E2 -29534.159} C_VEL
LIN {X 0,Y 92.085,Z 342.988,A -85,B 0,C 180,E1 -29538.918,E2 -29538.918} C_VEL
LIN {X 0,Y 92.072,Z 344.633,A -85,B 0,C 180,E1 -29539.178,E2 -29539.178} C_VEL
LIN {X 0,Y 88.664,Z 373.549,A -85,B 0,C 180,E1 -29540.486,E2 -29540.486} C_VEL
LIN {X 0,Y 85.89,Z 386.412,A -85,B 0,C 180,E1 -29541.463,E2 -29541.463} C_VEL
LIN {X 0,Y 82.126,Z 398.87,A -85,B 0,C 180,E1 -29543.065,E2 -29543.065} C_VEL
LIN {X 0,Y 77.548,Z 409.957,A -85,B 0,C 180,E1 -29544.987,E2 -29544.987} C_VEL
LIN {X 0,Y 71.742,Z 421.616,A -85,B 0,C 180,E1 -29548.139,E2 -29548.139} C_VEL
LIN {X 0,Y 66.222,Z 431.04,A -85,B 0,C 180,E1 -29551.877,E2 -29551.877} C_VEL
LIN {X 0,Y 60.869,Z 438.84,A -85,B 0,C 180,E1 -29556.06,E2 -29556.06} C_VEL
LIN {X 0,Y 54.886,Z 447.032,A -85,B 0,C 180,E1 -29562.569,E2 -29562.569} C_VEL
LIN {X 0,Y 48.708,Z 455.021,A -85,B 0,C 180,E1 -29572.161,E2 -29572.161} C_VEL
LIN {X 0,Y 44.832,Z 460.418,A -85,B 0,C 180,E1 -29581.932,E2 -29581.932} C_VEL
LIN {X 0,Y 42.028,Z 465.666,A -85,B 0,C 180,E1 -29595.458,E2 -29595.458} C_VEL
LIN {X 0,Y 41.347,Z 469.695,A -85,B 0,C 180,E1 -29609.985,E2 -29609.985} C_VEL
LIN {X 0,Y 41.615,Z 471.735,A -85,B 0,C 180,E1 -29619.707,E2 -29619.707} C_VEL
LIN {X 0,Y 45.089,Z 474.562,A -85,B 0,C 180,E1 -29637.863,E2 -29637.863} C_VEL
LIN {X 0,Y 48.207,Z 475.402,A -85,B 0,C 180,E1 -29645.656,E2 -29645.656} C_VEL
LIN {X 0,Y 52.058,Z 475.842,A -85,B 0,C 180,E1 -29652.439,E2 -29652.439} C_VEL
LIN {X 0,Y 61.705,Z 475.575,A -85,B 0,C 180,E1 -29662.853,E2 -29662.853} C_VEL
LIN {X 0,Y 72.845,Z 473.832,A -85,B 0,C 180,E1 -29670.245,E2 -29670.245} C_VEL
LIN {X 0,Y 83.455,Z 470.94,A -85,B 0,C 180,E1 -29675.079,E2 -29675.079} C_VEL
LIN {X 0,Y 94.264,Z 466.826,A -85,B 0,C 180,E1 -29678.722,E2 -29678.722} C_VEL
LIN {X 0,Y 103.933,Z 462.126,A -85,B 0,C 180,E1 -29681.186,E2 -29681.186} C_VEL
LIN {X 0,Y 115.47,Z 455.105,A -85,B 0,C 180,E1 -29683.438,E2 -29683.438} C_VEL
LIN {X 0,Y 125.444,Z 447.532,A -85,B 0,C 180,E1 -29685.091,E2 -29685.091} C_VEL
LIN {X 0,Y 133.87,Z 439.8,A -85,B 0,C 180,E1 -29686.2,E2 -29686.2} C_VEL
LIN {X 0,Y 143.225,Z 429.322,A -85,B 0,C 180,E1 -29687.206,E2 -29687.206} C_VEL
LIN {X 0,Y 150.876,Z 418.737,A -85,B 0,C 180,E1 -29687.993,E2 -29687.993} C_VEL
LIN {X 0,Y 157.715,Z 406.773,A -85,B 0,C 180,E1 -29688.6,E2 -29688.6} C_VEL
LIN {X 0,Y 159.068,Z 404.042,A -85,B 0,C 180,E1 -29688.707,E2 -29688.707} C_VEL
LIN {X 0,Y 159.655,Z 402.734,A -85,B 0,C 180,E1 -29689.144,E2 -29689.144} C_VEL
LIN {X 0,Y 159.7,Z 402.583,A -85,B 0,C 180,E1 -29689.852,E2 -29689.852} C_VEL
LIN {X 0,Y 159.601,Z 402.855,A -85,B 0,C 180,E1 -29690.549,E2 -29690.549} C_VEL
LIN {X 0,Y 153.827,Z 413.868,A -85,B 0,C 180,E1 -29691.084,E2 -29691.084} C_VEL
LIN {X 0,Y 146.419,Z 425.045,A -85,B 0,C 180,E1 -29691.862,E2 -29691.862} C_VEL
LIN {X 0,Y 138.113,Z 435.186,A -85,B 0,C 180,E1 -29692.832,E2 -29692.832} C_VEL
LIN {X 0,Y 128.852,Z 444.372,A -85,B 0,C 180,E1 -29694.054,E2 -29694.054} C_VEL
LIN {X 0,Y 118.226,Z 452.886,A -85,B 0,C 180,E1 -29695.7,E2 -29695.7} C_VEL
LIN {X 0,Y 107.242,Z 459.978,A -85,B 0,C 180,E1 -29697.829,E2 -29697.829} C_VEL
LIN {X 0,Y 98.29,Z 464.621,A -85,B 0,C 180,E1 -29699.984,E2 -29699.984} C_VEL
LIN {X 0,Y 87.964,Z 468.904,A -85,B 0,C 180,E1 -29703.067,E2 -29703.067} C_VEL
LIN {X 0,Y 76.649,Z 472.297,A -85,B 0,C 180,E1 -29707.689,E2 -29707.689} C_VEL
LIN {X 0,Y 71.466,Z 473.431,A -85,B 0,C 180,E1 -29709.752,E2 -29709.752} C_VEL
LIN {X 0,Y 62.175,Z 474.696,A -85,B 0,C 180,E1 -29712.547,E2 -29712.547} C_VEL
LIN {X 0,Y 54.791,Z 475.116,A -85,B 0,C 180,E1 -29715.373,E2 -29715.373} C_VEL
LIN {X 0,Y 49.775,Z 475.102,A -85,B 0,C 180,E1 -29718.801,E2 -29718.801} C_VEL
LIN {X 0,Y 48.313,Z 474.983,A -85,B 0,C 180,E1 -29720.341,E2 -29720.341} C_VEL
LIN {X 0,Y 41.188,Z 474.079,A -85,B 0,C 180,E1 -29731.472,E2 -29731.472} C_VEL
LIN {X 0,Y 37.319,Z 472.851,A -85,B 0,C 180,E1 -29741.15,E2 -29741.15} C_VEL
LIN {X 0,Y 34.403,Z 470.805,A -85,B 0,C 180,E1 -29754.717,E2 -29754.717} C_VEL
LIN {X 0,Y 33.56,Z 467.662,A -85,B 0,C 180,E1 -29771.712,E2 -29771.712} C_VEL
LIN {X 0,Y 35.632,Z 463.029,A -85,B 0,C 180,E1 -29790.018,E2 -29790.018} C_VEL
LIN {X 0,Y 40.08,Z 457.162,A -85,B 0,C 180,E1 -29805.266,E2 -29805.266} C_VEL
LIN {X 0,Y 46.359,Z 449.798,A -85,B 0,C 180,E1 -29817.067,E2 -29817.067} C_VEL
LIN {X 0,Y 54.083,Z 440.577,A -85,B 0,C 180,E1 -29825.801,E2 -29825.801} C_VEL
LIN {X 0,Y 61.139,Z 431.081,A -85,B 0,C 180,E1 -29831.387,E2 -29831.387} C_VEL
LIN {X 0,Y 67.898,Z 420.433,A -85,B 0,C 180,E1 -29835.38,E2 -29835.38} C_VEL
LIN {X 0,Y 73.915,Z 408.92,A -85,B 0,C 180,E1 -29838.304,E2 -29838.304} C_VEL
LIN {X 0,Y 78.811,Z 397.2,A -85,B 0,C 180,E1 -29840.288,E2 -29840.288} C_VEL
LIN {X 0,Y 82.98,Z 383.605,A -85,B 0,C 180,E1 -29841.835,E2 -29841.835} C_VEL
LIN {X 0,Y 85.696,Z 370.548,A -85,B 0,C 180,E1 -29842.733,E2 -29842.733} C_VEL
LIN {X 0,Y 88.578,Z 345.755,A -85,B 0,C 180,E1 -29843.842,E2 -29843.842} C_VEL
LIN {X 0,Y 86.623,Z 339.921,A -85,B 0,C 180,E1 -29848.182,E2 -29848.182} C_VEL
LIN {X 0,Y 84.67,Z 334.991,A -85,B 0,C 180,E1 -29853.53,E2 -29853.53} C_VEL
LIN {X 0,Y 83.882,Z 333.055,A -85,B 0,C 180,E1 -29856.349,E2 -29856.349} C_VEL
LIN {X 0,Y 82.812,Z 330.281,A -85,B 0,C 180,E1 -29861.972,E2 -29861.972} C_VEL
LIN {X 0,Y 82.31,Z 329.102,A -85,B 0,C 180,E1 -29870.187,E2 -29870.187} C_VEL
LIN {X 0,Y 82.886,Z 329.578,A -85,B 0,C 180,E1 -29876.781,E2 -29876.781} C_VEL
LIN {X 0,Y 83.542,Z 331.683,A -85,B 0,C 180,E1 -29880.795,E2 -29880.795} C_VEL
LIN {X 0,Y 84.314,Z 333.708,A -85,B 0,C 180,E1 -29883.953,E2 -29883.953} C_VEL
LIN {X 0,Y 86.246,Z 338.713,A -85,B 0,C 180,E1 -29889.663,E2 -29889.663} C_VEL
LIN {X 0,Y 88.165,Z 344.495,A -85,B 0,C 180,E1 -29894.137,E2 -29894.137} C_VEL
LIN {X 0,Y 88.633,Z 346.08,A -85,B 0,C 180,E1 -29895.13,E2 -29895.13} C_VEL
LIN {X 0,Y 85.458,Z 372.785,A -85,B 0,C 180,E1 -29896.331,E2 -29896.331} C_VEL
LIN {X 0,Y 82.588,Z 385.782,A -85,B 0,C 180,E1 -29897.176,E2 -29897.176} C_VEL
LIN {X 0,Y 78.795,Z 398.011,A -85,B 0,C 180,E1 -29898.592,E2 -29898.592} C_VEL
LIN {X 0,Y 74.027,Z 409.316,A -85,B 0,C 180,E1 -29900.339,E2 -29900.339} C_VEL
LIN {X 0,Y 68.676,Z 419.779,A -85,B 0,C 180,E1 -29902.902,E2 -29902.902} C_VEL
LIN {X 0,Y 62.735,Z 429.489,A -85,B 0,C 180,E1 -29906.313,E2 -29906.313} C_VEL
LIN {X 0,Y 56.923,Z 437.521,A -85,B 0,C 180,E1 -29910.181,E2 -29910.181} C_VEL
LIN {X 0,Y 51.584,Z 444.4,A -85,B 0,C 180,E1 -29915.149,E2 -29915.149} C_VEL
LIN {X 0,Y 44.365,Z 452.852,A -85,B 0,C 180,E1 -29924.512,E2 -29924.512} C_VEL
LIN {X 0,Y 38.683,Z 459.636,A -85,B 0,C 180,E1 -29936.953,E2 -29936.953} C_VEL
LIN {X 0,Y 35.202,Z 465.025,A -85,B 0,C 180,E1 -29952.555,E2 -29952.555} C_VEL
LIN {X 0,Y 34.267,Z 469.18,A -85,B 0,C 180,E1 -29969.982,E2 -29969.982} C_VEL
LIN {X 0,Y 34.66,Z 471.329,A -85,B 0,C 180,E1 -29981.68,E2 -29981.68} C_VEL
LIN {X 0,Y 38.951,Z 474.271,A -85,B 0,C 180,E1 -30002.752,E2 -30002.752} C_VEL
LIN {X 0,Y 47.049,Z 475.685,A -85,B 0,C 180,E1 -30018.301,E2 -30018.301} C_VEL
LIN {X 0,Y 57.682,Z 475.563,A -85,B 0,C 180,E1 -30028.505,E2 -30028.505} C_VEL
LIN {X 0,Y 69.591,Z 473.938,A -85,B 0,C 180,E1 -30035.333,E2 -30035.333} C_VEL
LIN {X 0,Y 80.062,Z 471.388,A -85,B 0,C 180,E1 -30039.424,E2 -30039.424} C_VEL
LIN {X 0,Y 91.935,Z 467.237,A -85,B 0,C 180,E1 -30042.832,E2 -30042.832} C_VEL
LIN {X 0,Y 101.875,Z 462.674,A -85,B 0,C 180,E1 -30044.948,E2 -30044.948} C_VEL
LIN {X 0,Y 113.662,Z 455.802,A -85,B 0,C 180,E1 -30046.845,E2 -30046.845} C_VEL
LIN {X 0,Y 123.82,Z 448.419,A -85,B 0,C 180,E1 -30048.241,E2 -30048.241} C_VEL
LIN {X 0,Y 132.369,Z 440.894,A -85,B 0,C 180,E1 -30049.158,E2 -30049.158} C_VEL
LIN {X 0,Y 135.805,Z 437.448,A -85,B 0,C 180,E1 -30049.474,E2 -30049.474} C_VEL
LIN {X 0,Y 135.545,Z 437.697,A -85,B 0,C 180,E1 -30050.083,E2 -30050.083} C_VEL
LIN {X 0,Y 126.249,Z 446.348,A -85,B 0,C 180,E1 -30051.119,E2 -30051.119} C_VEL
LIN {X 0,Y 117.003,Z 453.435,A -85,B 0,C 180,E1 -30052.306,E2 -30052.306} C_VEL
LIN {X 0,Y 105.979,Z 460.31,A -85,B 0,C 180,E1 -30054.048,E2 -30054.048} C_VEL
LIN {X 0,Y 94.19,Z 466.026,A -85,B 0,C 180,E1 -30056.448,E2 -30056.448} C_VEL
LIN {X 0,Y 84.336,Z 469.713,A -85,B 0,C 180,E1 -30059.03,E2 -30059.03} C_VEL
LIN {X 0,Y 73.158,Z 472.712,A -85,B 0,C 180,E1 -30062.978,E2 -30062.978} C_VEL
LIN {X 0,Y 63.795,Z 474.39,A -85,B 0,C 180,E1 -30067.558,E2 -30067.558} C_VEL
LIN {X 0,Y 53.142,Z 475.16,A -85,B 0,C 180,E1 -30075.306,E2 -30075.306} C_VEL
LIN {X 0,Y 48.313,Z 474.983,A -85,B 0,C 180,E1 -30080.341,E2 -30080.341} C_VEL
LIN {X 0,Y 43.862,Z 474.667,A -85,B 0,C 180,E1 -30085.134,E2 -30085.134} C_VEL
LIN {X 0,Y 35.956,Z 473.392,A -85,B 0,C 180,E1 -30093.551,E2 -30093.551} C_VEL
LIN {X 0,Y 30.296,Z 471.841,A -85,B 0,C 180,E1 -30102.92,E2 -30102.92} C_VEL
LIN {X 0,Y 27.457,Z 470.33,A -85,B 0,C 180,E1 -30112.865,E2 -30112.865} C_VEL
LIN {X 0,Y 26.962,Z 469.742,A -85,B 0,C 180,E1 -30116.744,E2 -30116.744} C_VEL
LIN {X 0,Y 27.171,Z 465.423,A -85,B 0,C 180,E1 -30142.6,E2 -30142.6} C_VEL
LIN {X 0,Y 31.159,Z 460.148,A -85,B 0,C 180,E1 -30163.056,E2 -30163.056} C_VEL
LIN {X 0,Y 37.516,Z 453.515,A -85,B 0,C 180,E1 -30177.945,E2 -30177.945} C_VEL
LIN {X 0,Y 45.439,Z 445.211,A -85,B 0,C 180,E1 -30188.237,E2 -30188.237} C_VEL
LIN {X 0,Y 52.817,Z 436.705,A -85,B 0,C 180,E1 -30194.329,E2 -30194.329} C_VEL
LIN {X 0,Y 59.811,Z 427.408,A -85,B 0,C 180,E1 -30198.526,E2 -30198.526} C_VEL
LIN {X 0,Y 66.236,Z 417.265,A -85,B 0,C 180,E1 -30201.508,E2 -30201.508} C_VEL
LIN {X 0,Y 71.907,Z 406.234,A -85,B 0,C 180,E1 -30203.754,E2 -30203.754} C_VEL
LIN {X 0,Y 76.853,Z 394.055,A -85,B 0,C 180,E1 -30205.402,E2 -30205.402} C_VEL
LIN {X 0,Y 80.741,Z 380.893,A -85,B 0,C 180,E1 -30206.596,E2 -30206.596} C_VEL
LIN {X 0,Y 83.269,Z 367.65,A -85,B 0,C 180,E1 -30207.26,E2 -30207.26} C_VEL
LIN {X 0,Y 85.499,Z 348.915,A -85,B 0,C 180,E1 -30207.988,E2 -30207.988} C_VEL
LIN {X 0,Y 84.097,Z 344.286,A -85,B 0,C 180,E1 -30211.961,E2 -30211.961} C_VEL
LIN {X 0,Y 82.704,Z 340.054,A -85,B 0,C 180,E1 -30217.141,E2 -30217.141} C_VEL
LIN {X 0,Y 81.801,Z 337.257,A -85,B 0,C 180,E1 -30222.572,E2 -30222.572} C_VEL
LIN {X 0,Y 81.401,Z 336.158,A -85,B 0,C 180,E1 -30230.076,E2 -30230.076} C_VEL
LIN {X 0,Y 81.895,Z 336.65,A -85,B 0,C 180,E1 -30236.365,E2 -30236.365} C_VEL
LIN {X 0,Y 82.8,Z 340.063,A -85,B 0,C 180,E1 -30242.002,E2 -30242.002} C_VEL
LIN {X 0,Y 84.347,Z 344.805,A -85,B 0,C 180,E1 -30247.555,E2 -30247.555} C_VEL
LIN {X 0,Y 85.519,Z 349.013,A -85,B 0,C 180,E1 -30250.898,E2 -30250.898} C_VEL
LIN {X 0,Y 83.693,Z 365.143,A -85,B 0,C 180,E1 -30251.591,E2 -30251.591} C_VEL
LIN {X 0,Y 81.533,Z 378.042,A -85,B 0,C 180,E1 -30252.106,E2 -30252.106} C_VEL
LIN {X 0,Y 78.036,Z 391.155,A -85,B 0,C 180,E1 -30253.116,E2 -30253.116} C_VEL
LIN {X 0,Y 73.528,Z 403.31,A -85,B 0,C 180,E1 -30254.555,E2 -30254.555} C_VEL
LIN {X 0,Y 67.782,Z 414.917,A -85,B 0,C 180,E1 -30256.415,E2 -30256.415} C_VEL
LIN {X 0,Y 62.22,Z 424.338,A -85,B 0,C 180,E1 -30258.887,E2 -30258.887} C_VEL
LIN {X 0,Y 56.13,Z 433.097,A -85,B 0,C 180,E1 -30262.2,E2 -30262.2} C_VEL
LIN {X 0,Y 49.297,Z 441.551,A -85,B 0,C 180,E1 -30266.971,E2 -30266.971} C_VEL
LIN {X 0,Y 41.005,Z 450.585,A -85,B 0,C 180,E1 -30275.474,E2 -30275.474} C_VEL
LIN {X 0,Y 33.925,Z 457.815,A -85,B 0,C 180,E1 -30287.655,E2 -30287.655} C_VEL
LIN {X 0,Y 29.66,Z 462.683,A -85,B 0,C 180,E1 -30301.688,E2 -30301.688} C_VEL
LIN {X 0,Y 27.226,Z 467.366,A -85,B 0,C 180,E1 -30322.561,E2 -30322.561} C_VEL
LIN {X 0,Y 27.274,Z 469.826,A -85,B 0,C 180,E1 -30337.379,E2 -30337.379} C_VEL
LIN {X 0,Y 29.807,Z 472.636,A -85,B 0,C 180,E1 -30358.112,E2 -30358.112} C_VEL
LIN {X 0,Y 37.559,Z 474.919,A -85,B 0,C 180,E1 -30378.432,E2 -30378.432} C_VEL
LIN {X 0,Y 48.314,Z 475.719,A -85,B 0,C 180,E1 -30390.757,E2 -30390.757} C_VEL
LIN {X 0,Y 60.524,Z 474.981,A -85,B 0,C 180,E1 -30398.243,E2 -30398.243} C_VEL
LIN {X 0,Y 73.456,Z 472.724,A -85,B 0,C 180,E1 -30403.059,E2 -30403.059} C_VEL
LIN {X 0,Y 83.381,Z 469.971,A -85,B 0,C 180,E1 -30405.736,E2 -30405.736} C_VEL
LIN {X 0,Y 93.474,Z 466.241,A -85,B 0,C 180,E1 -30407.768,E2 -30407.768} C_VEL
LIN {X 0,Y 103.697,Z 461.429,A -85,B 0,C 180,E1 -30409.299,E2 -30409.299} C_VEL
LIN {X 0,Y 107.108,Z 459.579,A -85,B 0,C 180,E1 -30409.779,E2 -30409.779} C_VEL
LIN {X 0,Y 107.048,Z 459.609,A -85,B 0,C 180,E1 -30409.958,E2 -30409.958} C_VEL
LIN {X 0,Y 96.106,Z 465.068,A -85,B 0,C 180,E1 -30411.574,E2 -30411.574} C_VEL
LIN {X 0,Y 84.823,Z 469.377,A -85,B 0,C 180,E1 -30413.784,E2 -30413.784} C_VEL
LIN {X 0,Y 77.526,Z 471.507,A -85,B 0,C 180,E1 -30415.59,E2 -30415.59} C_VEL
LIN {X 0,Y 64.494,Z 474.172,A -85,B 0,C 180,E1 -30419.976,E2 -30419.976} C_VEL
LIN {X 0,Y 56.347,Z 475.02,A -85,B 0,C 180,E1 -30423.958,E2 -30423.958} C_VEL
LIN {X 0,Y 49.706,Z 475.278,A -85,B 0,C 180,E1 -30428.303,E2 -30428.303} C_VEL
LIN {X 0,Y 43.427,Z 475.046,A -85,B 0,C 180,E1 -30433.892,E2 -30433.892} C_VEL
LIN {X 0,Y 37.128,Z 474.26,A -85,B 0,C 180,E1 -30442.2,E2 -30442.2} C_VEL
LIN {X 0,Y 32.751,Z 473.235,A -85,B 0,C 180,E1 -30450.906,E2 -30450.906} C_VEL
LIN {X 0,Y 27.951,Z 470.868,A -85,B 0,C 180,E1 -30468.878,E2 -30468.878} C_VEL
LIN {X 0,Y 26.962,Z 469.742,A -85,B 0,C 180,E1 -30476.744,E2 -30476.744} C_VEL
LIN {X 0,Y 25.772,Z 467.921,A -85,B 0,C 180,E1 -30488.675,E2 -30488.675} C_VEL
LIN {X 0,Y 24.709,Z 465.808,A -85,B 0,C 180,E1 -30501.071,E2 -30501.071} C_VEL
LIN {X 0,Y 25.771,Z 459.903,A -85,B 0,C 180,E1 -30530.088,E2 -30530.088} C_VEL
LIN {X 0,Y 28.597,Z 456.88,A -85,B 0,C 180,E1 -30539.345,E2 -30539.345} C_VEL
LIN {X 0,Y 37.148,Z 449.154,A -85,B 0,C 180,E1 -30551.992,E2 -30551.992} C_VEL
LIN {X 0,Y 46.316,Z 439.996,A -85,B 0,C 180,E1 -30559.37,E2 -30559.37} C_VEL
LIN {X 0,Y 54.439,Z 430.271,A -85,B 0,C 180,E1 -30563.81,E2 -30563.81} C_VEL
LIN {X 0,Y 61.979,Z 419.417,A -85,B 0,C 180,E1 -30566.766,E2 -30566.766} C_VEL
LIN {X 0,Y 68.621,Z 407.472,A -85,B 0,C 180,E1 -30568.907,E2 -30568.907} C_VEL
LIN {X 0,Y 73.897,Z 395.174,A -85,B 0,C 180,E1 -30570.315,E2 -30570.315} C_VEL
LIN {X 0,Y 78.011,Z 382.14,A -85,B 0,C 180,E1 -30571.315,E2 -30571.315} C_VEL
LIN {X 0,Y 80.691,Z 369.066,A -85,B 0,C 180,E1 -30571.894,E2 -30571.894} C_VEL
LIN {X 0,Y 82.803,Z 352.113,A -85,B 0,C 180,E1 -30572.501,E2 -30572.501} C_VEL
LIN {X 0,Y 81.612,Z 347.658,A -85,B 0,C 180,E1 -30577.441,E2 -30577.441} C_VEL
LIN {X 0,Y 80.979,Z 345.43,A -85,B 0,C 180,E1 -30581.225,E2 -30581.225} C_VEL
LIN {X 0,Y 80.704,Z 344.097,A -85,B 0,C 180,E1 -30584.023,E2 -30584.023} C_VEL
LIN {X 0,Y 80.555,Z 343.18,A -85,B 0,C 180,E1 -30591.866,E2 -30591.866} C_VEL
LIN {X 0,Y 80.833,Z 343.637,A -85,B 0,C 180,E1 -30595.353,E2 -30595.353} C_VEL
LIN {X 0,Y 81.546,Z 347.008,A -85,B 0,C 180,E1 -30600.864,E2 -30600.864} C_VEL
LIN {X 0,Y 82.758,Z 351.776,A -85,B 0,C 180,E1 -30606.112,E2 -30606.112} C_VEL
LIN {X 0,Y 82.846,Z 352.199,A -85,B 0,C 180,E1 -30606.449,E2 -30606.449} C_VEL
LIN {X 0,Y 81.441,Z 364.221,A -85,B 0,C 180,E1 -30606.947,E2 -30606.947} C_VEL
LIN {X 0,Y 79.276,Z 377.226,A -85,B 0,C 180,E1 -30607.3,E2 -30607.3} C_VEL
LIN {X 0,Y 75.878,Z 389.951,A -85,B 0,C 180,E1 -30608.095,E2 -30608.095} C_VEL
LIN {X 0,Y 71.215,Z 402.358,A -85,B 0,C 180,E1 -30609.246,E2 -30609.246} C_VEL
LIN {X 0,Y 65.275,Z 414.202,A -85,B 0,C 180,E1 -30610.697,E2 -30610.697} C_VEL
LIN {X 0,Y 59.455,Z 423.733,A -85,B 0,C 180,E1 -30612.739,E2 -30612.739} C_VEL
LIN {X 0,Y 52.942,Z 432.681,A -85,B 0,C 180,E1 -30615.562,E2 -30615.562} C_VEL
LIN {X 0,Y 46.488,Z 440.258,A -85,B 0,C 180,E1 -30619.075,E2 -30619.075} C_VEL
LIN {X 0,Y 37.319,Z 449.509,A -85,B 0,C 180,E1 -30626.514,E2 -30626.514} C_VEL
LIN {X 0,Y 29.038,Z 456.916,A -85,B 0,C 180,E1 -30638.097,E2 -30638.097} C_VEL
LIN {X 0,Y 23.637,Z 461.933,A -85,B 0,C 180,E1 -30653.48,E2 -30653.48} C_VEL
LIN {X 0,Y 20.216,Z 466.757,A -85,B 0,C 180,E1 -30679.958,E2 -30679.958} C_VEL
LIN {X 0,Y 20.278,Z 469.32,A -85,B 0,C 180,E1 -30699.948,E2 -30699.948} C_VEL
LIN {X 0,Y 23.794,Z 472.227,A -85,B 0,C 180,E1 -30726.175,E2 -30726.175} C_VEL
LIN {X 0,Y 28.074,Z 473.665,A -85,B 0,C 180,E1 -30738.643,E2 -30738.643} C_VEL
LIN {X 0,Y 39.058,Z 475.315,A -85,B 0,C 180,E1 -30754.08,E2 -30754.08} C_VEL
LIN {X 0,Y 51.687,Z 475.5,A -85,B 0,C 180,E1 -30762.099,E2 -30762.099} C_VEL
LIN {X 0,Y 58.267,Z 475.026,A -85,B 0,C 180,E1 -30764.74,E2 -30764.74} C_VEL
LIN {X 0,Y 71.706,Z 472.886,A -85,B 0,C 180,E1 -30768.506,E2 -30768.506} C_VEL
LIN {X 0,Y 74.42,Z 472.301,A -85,B 0,C 180,E1 -30769.092,E2 -30769.092} C_VEL
LIN {X 0,Y 75.126,Z 472.1,A -85,B 0,C 180,E1 -30770.586,E2 -30770.586} C_VEL
LIN {X 0,Y 63.248,Z 474.314,A -85,B 0,C 180,E1 -30773.596,E2 -30773.596} C_VEL
LIN {X 0,Y 56.352,Z 475.028,A -85,B 0,C 180,E1 -30775.969,E2 -30775.969} C_VEL
LIN {X 0,Y 47.85,Z 475.38,A -85,B 0,C 180,E1 -30779.967,E2 -30779.967} C_VEL
LIN {X 0,Y 35.615,Z 474.632,A -85,B 0,C 180,E1 -30789.475,E2 -30789.475} C_VEL
LIN {X 0,Y 29.526,Z 473.577,A -85,B 0,C 180,E1 -30797.877,E2 -30797.877} C_VEL
LIN {X 0,Y 21.847,Z 470.895,A -85,B 0,C 180,E1 -30819.949,E2 -30819.949} C_VEL
LIN {X 0,Y 19.36,Z 467.559,A -85,B 0,C 180,E1 -30848.749,E2 -30848.749} C_VEL
LIN {X 0,Y 22.414,Z 462.559,A -85,B 0,C 180,E1 -30880.509,E2 -30880.509} C_VEL
LIN {X 0,Y 28.597,Z 456.88,A -85,B 0,C 180,E1 -30899.345,E2 -30899.345} C_VEL
LIN {X 0,Y 31.795,Z 453.736,A -85,B 0,C 180,E1 -30906.649,E2 -30906.649} C_VEL
LIN {X 0,Y 36.552,Z 448.047,A -85,B 0,C 180,E1 -30917.72,E2 -30917.72} C_VEL
LIN {X 0,Y 41.843,Z 441.74,A -85,B 0,C 180,E1 -30925.899,E2 -30925.899} C_VEL
LIN {X 0,Y 45.556,Z 437.596,A -85,B 0,C 180,E1 -30928.628,E2 -30928.628} C_VEL
LIN {X 0,Y 53.95,Z 427.631,A -85,B 0,C 180,E1 -30931.582,E2 -30931.582} C_VEL
LIN {X 0,Y 60.941,Z 417.489,A -85,B 0,C 180,E1 -30933.372,E2 -30933.372} C_VEL
LIN {X 0,Y 67.198,Z 406.111,A -85,B 0,C 180,E1 -30934.809,E2 -30934.809} C_VEL
LIN {X 0,Y 72.501,Z 393.725,A -85,B 0,C 180,E1 -30935.791,E2 -30935.791} C_VEL
LIN {X 0,Y 76.466,Z 380.912,A -85,B 0,C 180,E1 -30936.455,E2 -30936.455} C_VEL
LIN {X 0,Y 79.156,Z 367.3,A -85,B 0,C 180,E1 -30936.839,E2 -30936.839} C_VEL
LIN {X 0,Y 80.592,Z 355.822,A -85,B 0,C 180,E1 -30937.246,E2 -30937.246} C_VEL
LIN {X 0,Y 80.013,Z 352.815,A -85,B 0,C 180,E1 -30941.244,E2 -30941.244} C_VEL
LIN {X 0,Y 79.66,Z 350.898,A -85,B 0,C 180,E1 -30945.582,E2 -30945.582} C_VEL
LIN {X 0,Y 79.643,Z 350.225,A -85,B 0,C 180,E1 -30951.772,E2 -30951.772} C_VEL
LIN {X 0,Y 79.801,Z 350.678,A -85,B 0,C 180,E1 -30954.405,E2 -30954.405} C_VEL
LIN {X 0,Y 80.195,Z 353.352,A -85,B 0,C 180,E1 -30958.801,E2 -30958.801} C_VEL
LIN {X 0,Y 80.66,Z 355.832,A -85,B 0,C 180,E1 -30961.812,E2 -30961.812} C_VEL
